// TwinCAT 3 PLC project Library
// Title: PMPS
// Company: SLAC - LCLS
// Author: Alex Wallace and contributors
// ProjectVersion: 0.0.0
// Description: Collection of PMPS functionality for LCLS PLCs
// ProgramVersion: 3.1.4023.0
// libraries:
//   Tc2_MC2, * (Beckhoff Automation GmbH)
//   Tc2_Standard, * (Beckhoff Automation GmbH)
//   Tc2_System, * (Beckhoff Automation GmbH)
//   Tc2_Utilities, * (Beckhoff Automation GmbH)
//   Tc3_JsonXml, * (Beckhoff Automation GmbH)
//   Tc3_Module, * (Beckhoff Automation GmbH)
//   LCLS General,newest,SLAC
//   TcUnit,newest,www.tcunit.org
// project tree:
//   DUTs/ E_BPTMState.TcDUT, K_Apertures.TcTLEO (not stored), L_Apertures.TcTLEO (not stored), L_Stopper.TcTLEO, K_Stopper.TcTLEO (not stored), ST_BeamParams_WC.TcDUT, ST_BeamParams.TcDUT, ST_Device.TcDUT (not stored), ST_DeviceState.TcDUT, ST_DeviceStateExt.TcDUT (not stored), ST_DeviceStateTable.TcDUT, ST_FFInfo.TcDUT, ST_FF.TcDUT, ST_FFOverride.TcDUT, ST_PMPS_Aperture.TcDUT, ST_PMPS_Attenuator.TcDUT, T_HashTableEntry.TcDUT (not stored)
//   GVLs/ PMPS_GVL.TcGVL
//   HelperFunctions/ APT_TO_IO.TcPOU (not stored), ATT_TO_IO.TcPOU (not stored), F_DeviceState_To_DeviceStateExt.TcPOU (not stored), F_DifferentBeamParams.TcPOU, F_eVRangeCalculator.TcPOU (not stored), F_eVWithinSpec.TcPOU, F_SafeBPCompare.TcPOU, F_SetBeamParams.TcPOU, F_SetStateParams.TcPOU (not stored), IO_TO_APT.TcPOU (not stored), IO_TO_ATT.TcPOU, IO_TO_BP.TcPOU, BP_TO_IO.TcPOU
//   / MAIN.TcPOU, PlcTask.TcTTO (not stored)
//   MajorComponents/Arbiter/ FB_Arbiter.TcPOU, FB_BeamParamAssertionPool.TcPOU
//   MajorComponents/ BeamParameterTransitionManager.TcPOU, FB_BPRequestor.TcPOU, FB_LinearDeviceStateTable.TcPOU, FB_LinearGovernor.TcPOU, I_HigherAuthority.TcIO
//   MajorComponents/FastFaults/ FB_FastFault.TcPOU, FB_FastFaultLogger.TcPOU, FB_HardwareFFOutput.TcPOU
//   MajorComponents/InterPlcComm/ FB_ArbiterToSubSys_IO.TcPOU, FB_SubSysToArbiter_IO.TcPOU
//   MajorComponents/PMPS_MPS_Interface/ FB_BeamClassOutputs.TcPOU, FB_CTLS_Outputs.TcPOU, FB_PhotonEnergyWatcher.TcPOU
//   TestComponents/ eBPTMTestStates.TcDUT (not stored), FB_Arbiter_Test.TcPOU, FB_AttenuatorSimulator.TcPOU (not stored), FB_BPTM_Test.TcPOU, FB_ArbToSubsys_Test.TcPOU, FB_DiffBP_Test.TcPOU (not stored), FB_SubsysToArb_Test.TcPOU, FB_evRangeCalculator_Test.TcPOU, FB_eVWithinSpec_Test.TcPOU (not stored), FB_FastFault_Test.TcPOU, FB_MachineSimulator.TcPOU, FB_PhotonEnergyWatcher_Test.TcPOU, FB_SafeBPCompare_Test.TcPOU, FB_SolidAttenuator.TcPOU (not stored) (excluded from build)
// real-time tasks:
//   TASK PlcTask: cycle T#10ms, priority 20, ADS port 350

// ---- DUTs/E_BPTMState.TcDUT
TYPE E_BPTMState :
(
	NewTarget := 1,
    WaitingForTransitionAssertion := 2,
    WaitingForFinalAssertion := 3,
    Transitioning := 4,
    CleaningUp := 5
);
END_TYPE

// ---- DUTs/L_Stopper.TcTLEO
{attribute 'qualified_only'}
{attribute 'strict'}
TYPE L_Stopper :
(
	ST1 := 1,
    ST2 := 2
);
END_TYPE

// ---- DUTs/ST_BeamParams_WC.TcDUT
TYPE ST_BeamParams_WC : 
    STRUCT
        (*  Requested pre-optic attenuation %  *)
		{attribute 'pytmc' := 'pv: Attenuation
        io: i'}
		fAtt : REAL := 100;
        (* Pulse-rate *)
        {attribute 'pytmc' := 'pv: Rate
        io: i'}
        nRate : UDINT := 10;
        (* Per pulse max energy (mJ) *)
        {attribute 'pytmc' := 'pv: PulseEnergy
        io: i'}
        fPP_mJ : REAL := 20;
        (* Photon energy ranges *)
        {attribute 'pytmc' := 'pv: PhotonEnergy
        io: i'}
        {attribute 'displaymode' := 'binary'}
        neVRange : WORD := 65535;
        (* Beamline attenuators *)
        {attribute 'pytmc' := 'pv: AuxAttenuator
        io: i'}
        astAttenuators : ARRAY [1..32] OF ST_PMPS_Attenuator;
        // Toggle for watchdog
        xValidToggle : BOOL;
        // Beam parameter set is valid (if readback), or acknowledged (if request)
        {attribute 'pytmc' := 'pv: Valid
        io: i'}
        xValid : BOOL;
        // Cohort index. Identifies which cohort this BP set was included in arbitration
        {attribute 'pytmc' := 'pv: Attenuation
        io: i'}
        nCohortInt : ULINT;
    END_STRUCT
END_TYPE

// ---- DUTs/ST_BeamParams.TcDUT
TYPE ST_BeamParams : 
    STRUCT
        (*  Requested pre-optic attenuation %  *)
		{attribute 'pytmc' := 'pv: Attenuation
            io: i
            field: EGU %
        '}
		fAtt : REAL := 100;
        (* Pulse-rate *)
        {attribute 'pytmc' := 'pv: Rate
            io: i
            field: EGU Hz
        '}
        nRate : UDINT := 10;
        (* Per pulse max energy (mJ) *)
        {attribute 'pytmc' := 'pv: PulseEnergy
            io: i
            field: EGU mJ
        '}
        fPP_mJ : REAL := 20;
        (* Photon energy ranges *)
        {attribute 'pytmc' := 'pv: PhotonEnergyRanges
            io: i
            field: EGU eV'}
        {attribute 'displaymode' := 'binary'}
        neVRange : WORD := 65535;
        (* Beamline attenuators *)
        {attribute 'pytmc' := 'pv: AuxAtt
        io: i'}
        astAttenuators : ARRAY [1..PMPS_GVL.AUX_ATTENUATORS] OF ST_PMPS_Attenuator;
        
        (* Stoppers *)
        {attribute 'pytmc' := 'pv: ST
        io: i'}
        aStoppers : ARRAY [1..PMPS_GVL.MAX_STOPPERS] OF BOOL;
        
        (* Apertures *)
        astApertures : ARRAY [1..PMPS_GVL.MAX_APERTURES] OF ST_PMPS_Aperture;
        
        // Toggle for watchdog
        xValidToggle : BOOL;
        // Beam parameter set is valid (if readback), or acknowledged (if request)
        {attribute 'pytmc' := 'pv: Valid
        io: i'}
        xValid : BOOL;
        // Cohort index. Identifies which cohort this BP set was included in arbitration
        {attribute 'pytmc' := 'pv: Cohort
        io: i
            field: DESC Cohort inc on each arb cycle
        '}
        nCohortInt : UDINT;
    END_STRUCT
END_TYPE

// ---- DUTs/ST_DeviceState.TcDUT
TYPE ST_DeviceState :
STRUCT
	
	//State name
	sStateName	:	STRING;
	nStateRef	:	UDINT; //Primary key of device state database
	
	//////////////////
	// This stuff may belong in a sub-class or something
	//Position
	rPosition	:	REAL := 0; //Center of the state
	//Tolerance
	rTolerance :	REAL := 0; //+/- amount
	//////////////////
	//Required beam parameters
	stReqBeamParam	:	ST_BeamParams;

END_STRUCT
END_TYPE

// ---- DUTs/ST_DeviceStateTable.TcDUT
TYPE ST_DeviceStateTable :
STRUCT
	iDeviceID:DINT;
	iStateID:DINT;
	rTargetPosition: REAL;
	rTolerance: REAL;
	rTransmission: REAL;
	iBeamClass : DINT;
	iPulseRate: DINT;
	rPerPulseEnergy:REAL;
	rUpper_eV: REAL;
	rLower_eV: REAL;
	rPhotonEnergy: REAL;
END_STRUCT
END_TYPE

// ---- DUTs/ST_FFInfo.TcDUT

// These elements should be set at init and never changed.

TYPE ST_FFInfo :
STRUCT
    sPath   :    T_MaxString; // Full PLC path to FF object
    Desc    :   T_MaxString; // Set at instantiation to a helpful description of the fast fault purpose
    DevName :   T_MaxString; // Component name, used in diagnostic to help narrow down where beam faults are coming from
    TypeCode    :   UINT; // Set at instantiation to fault class code

///////////////////////////////////////////
// Warning, this variable is effectively a VETO of the fast fault if set FALSE
// Do not alter the state of this variable unless you really know what you're doing.
///////////////////////////////////////////
    InUse   :   BOOL := FALSE; // If this FF is currently in-use
///////////////////////////////////////////

 
    AutoReset   :   BOOL; // Automatically clear fast fault (latching vs non-latching)
    
    {attribute 'pytmc' := '
        pv: InfoString
        io: i
     '}
    InfoString : STRING;
END_STRUCT
END_TYPE

// ---- DUTs/ST_FF.TcDUT
TYPE ST_FF :
STRUCT
    {attribute 'pytmc' := '
        pv: Info
     '}
    Info : ST_FFInfo;
    
    {attribute 'pytmc' := '
        pv: Veto
     '}
    Veto : ST_FFVeto;
    
    {attribute 'pytmc' := '
        pv: OK
        io: i
     '}
    OK   :   BOOL; // Fault logic state
    
    FaultAck : BOOL; // Set when faulted, reset by logger.
    
    {attribute 'pytmc' := '
        pv: BeamPermitted
        io: i
     '}
    BeamPermitted   :   BOOL; // Result of reset, veto, and fault logic, true beam off boolean
    
    {attribute 'pytmc' := '
        pv: Reset
        io: o
     '}
    Reset   :   BOOL;
    
    bsFF    :    RS;
    rtReset    :    R_TRIG;
    ftCountFault : F_TRIG;
    
END_STRUCT
END_TYPE

// ---- DUTs/ST_FFOverride.TcDUT
TYPE ST_FFOverride :
STRUCT
    {attribute 'pytmc' := '
        pv: Duration
        io: o
     '}
    Duration : UDINT; // UDINT to be compatible with ESS module.
    
    {attribute 'pytmc' := '
        pv: Activate
        io: o
     '}
    Activate : BOOL;
    
    {attribute 'pytmc' := '
        pv: Deactivate
        io: o
     '}
    Deactivate : BOOL;
    
    {attribute 'pytmc' := '
        pv: ElapsedTime
        io: i
     '}
    ElapsedTime : UDINT; // UDINT to be compatible with ESS module.
    
    {attribute 'pytmc' := '
        pv: Active
        io: i
     '} 
	Active: BOOL;
    
    Timer    :   TP;
    OvrdActLogAck : BOOL;
    OvrdExpLogAck : BOOL;
    
    tOvrdActivate : R_TRIG;
    tOvrdExpiring  : F_TRIG;
END_STRUCT
END_TYPE

// ---- DUTs/ST_PMPS_Aperture.TcDUT
TYPE ST_PMPS_Aperture :
STRUCT
    {attribute 'pytmc' := 'pv: Width
            io: i
            field: EGU mm'}
    Width : REAL; // distance between horizontal slits (x)
    {attribute 'pytmc' := 'pv: Height
            io: i
            field: EGU mm'}
    Height : REAL; // distance between vertical slits (y)
    
    {attribute 'pytmc' := 'pv: OK
        io: i'}
    xOK : BOOL; // status of aperture, false if error or in motion
END_STRUCT
END_TYPE

// ---- DUTs/ST_PMPS_Attenuator.TcDUT
TYPE ST_PMPS_Attenuator EXTENDS ST_PMPS_Attenuator_IO :
STRUCT
    (*
        {attribute 'pytmc' := 'pv: Att
            io: i
            field: EGU %
        '}
		nAtt : UINT;
        {attribute 'pytmc' := 'pv: OK
            io: i
        '}
		xAttOK : UINT; // true = no errors and attenuator is stable
        *)
END_STRUCT
END_TYPE

// ---- GVLs/PMPS_GVL.TcGVL
{attribute 'qualified_only'}
VAR_GLOBAL
    {attribute 'pytmc' := '
        pv: @(PREFIX)RequestedBP
        archive: 1Hz monitor
    '}
    stRequestedBeamParameters    :    ST_BeamParams; //Summarized request for the line, as recognized by the line arbiter PLC
    {attribute 'pytmc' := '
        pv: @(PREFIX)CurrentBP
        archive: 1Hz monitor
    '}
    stCurrentBeamParameters    :    ST_BeamParams; //Currently active BP set, broadcast by the line arbiter PLC
    
    fbLog : FB_LogMessage:=(eSubsystem:=E_Subsystem.MPS);
END_VAR
VAR_GLOBAL RETAIN    
    // Statistics
    {attribute 'pytmc' := '
        pv: @(PREFIX)SuccessfulPreemptions
        io: i
    '}
    SuccessfulPreemption : UDINT; // Any time BPTM applies a new BP request which is confirmed
    {attribute 'pytmc' := '
        pv: @(PREFIX)AccumulatedFastFaults
        io: i
    '}
    AccumulatedFF : UDINT; // Any time a FF occurs
END_VAR
VAR_GLOBAL CONSTANT
    EXCLUDED_ASSERTION_ID    :    UDINT    := 16#FFFFFFFF; //An assertion ID that should always return "not found" in the assertion pool
    VISIBLE_TEST_VELOCITY    :    LREAL    := 10;
    FAST_TEST_VELOCITY        :    LREAL    := 100;
    MAX_DEVICE_STATES        :    UDINT    := 300;
    MAX_FAST_FAULTS : UINT := 50; // Maximum number of fast faults that can be associated with a FFO
    MAX_STOPPERS    :   UINT := 16;
    {attribute 'pytmc' := '
        pv: @(PREFIX)FullBeamCnst
        archive: 1Hz monitor
        field: DESC Full beam constant
    '}    
    cstFullBeam    :    ST_BeamParams := (
        fAtt := 0,
        fPP_mJ := 1E4,
        neVRange := 2#1111_1111_1111_1111,
        nRate    := UDINT#1000000
    );
    {attribute 'pytmc' := '
        pv: @(PREFIX)SafeBeamCnst
        archive: 1Hz monitor
        field: DESC Safe beam constant
    '} 
    cstSafeBeam    :    ST_BeamParams := (
        fAtt := 100,
        fPP_mJ := 0,
        neVRange := 0,
        nRate    := 0
    );
    cnMaxStateArrayLen : INT := 20;
    
    AUX_ATTENUATORS : UINT := 16; // Maximum # of attenuators in the PMPS
    MAX_APERTURES : UINT := 4; // Maximum # of power slits in the PMPS
    DUMMY_AUX_ATT_ARRAY : ARRAY [1..PMPS_GVL.AUX_ATTENUATORS] OF ST_PMPS_Attenuator;
    
    MAX_ASSERTIONS    :    UDINT := 20; //Maximum number of assertions permitted in the arbiter
    
    g_cBoundaries    :    INT    := 15;
    {attribute 'pytmc' := '
        pv: @(PREFIX)eVRangeCnst
        archive: 1Hz monitor
        field: DESC eV Range constants
        field: EGU keV
    '}
    g_areVBoundaries    :    ARRAY [0..g_cBoundaries]    OF    REAL    := [ 
    0.2,
    0.3,
    0.4,
    0.5,
    0.6,
    0.7,
    0.8,
    0.9,
    1.0,
    1.1,
    1.2,
    1.3,
    1.4,
    1.5,
    1.6,
    1.7
];


END_VAR

// ---- MajorComponents/I_HigherAuthority.TcIO
INTERFACE I_HigherAuthority

METHOD CheckRequest : BOOL
VAR_INPUT
    nReqID    :    DWORD;
END_VAR
END_METHOD

METHOD RequestBP : BOOL
VAR_INPUT
    nReqID    :    DWORD; //StateID of state requesting beam parameter set
    stReqBP        :    ST_BeamParams; //Requested beam params
END_VAR
END_METHOD

END_INTERFACE

// ---- HelperFunctions/F_DifferentBeamParams.TcPOU
{attribute 'obsolete' := 'Use Req and Readback BP structs instead.'} 
(*DEPRECATED Compares BeamParam1 to BeamParam2, if any parameters of BeamParam1 are different than BeamParam2
the result will be true. *)
FUNCTION F_DifferentBeamParams : BOOL
VAR_INPUT
    BeamParam1    :    ST_BeamParams;
    BeamParam2    :    ST_BeamParams;
END_VAR
VAR
    // Internal Attenuation OK boolean
    xAttOK: BOOL := FALSE;
    // Internal Per-pulse energy OK boolean
    xPPmjOK: BOOL := FALSE;
    // Internal photon energy OK boolean
    xEvOK: BOOL := FALSE;
    xRateOK: BOOL;
END_VAR

xAttOK := BeamParam1.fAtt <> BeamParam2.fAtt;
xPPmjOK := BeamParam1.fPP_mJ <> BeamParam2.fPP_mJ;
xEvOK := BeamParam1.neVRange <> BeamParam2.neVRange;
xRateOK     := BeamParam1.nRate <> BeamParam2.nRate;


F_DifferentBeamParams := xAttOK OR xPPmjOK OR xEvOK OR xRateOK;

END_FUNCTION

// ---- HelperFunctions/F_eVWithinSpec.TcPOU
//reV must be within permitted range.
FUNCTION F_eVWithinSpec : BOOL
VAR_INPUT
    reV    :    REAL;    //Photon energy to check if within permitted range
    nPermittedRange    :    WORD; //Permitted range
END_VAR
VAR
    //Holding register for permitted ranges
    nPermittedRangeHolding    :    WORD; 
    //For loop counter
    nIndex    :    INT;
    // Lower boundary for range check 
    rPreviousBoundary: REAL := 0;
END_VAR

(* How this works:
The within range bool is initialized to false.
Load the word representation of ranges into a holding register.
If the bit at position zero of the holding register is true, and the input eV is
below the boundary at the index position of the boundary array, and the previous boundary
(which initializes at 0), then the within range bool is set. 
Then, we stash the upper boundary as the lower boundary for the next comparison,
and shift the holding register right, which moves the next bit to the zero position.
*)
nPermittedRangeHolding := nPermittedRange;

FOR nIndex := 0 TO PMPS_GVL.g_cBoundaries DO
        
    F_eVWithinSpec S= nPermittedRangeHolding.0 AND( 
        (reV <= PMPS_GVL.g_areVBoundaries[nIndex]*1000) AND
        (reV >= rPreviousBoundary*1000) );
        
    IF F_eVWithinSpec THEN RETURN; END_IF
    
    rPreviousBoundary := PMPS_GVL.g_areVBoundaries[nIndex];
    nPermittedRangeHolding := SHR(nPermittedRangeHolding, 1);
END_FOR

END_FUNCTION

// ---- HelperFunctions/F_SafeBPCompare.TcPOU
(*Compares BeamParam1 to BeamParam2: if the parameters of BeamParam1 are more conservative than BeamParam2
the result will be true. *)
FUNCTION F_SafeBPCompare : BOOL
VAR_INPUT
    BeamParam1    :    ST_BeamParams; //Must be more conservative than 2
    BeamParam2    :    ST_BeamParams;
END_VAR
VAR
    // Internal Attenuation OK boolean
    xAttOK: BOOL := FALSE;
    // Internal Per-pulse energy OK boolean
    xPPmjOK: BOOL := FALSE;
    // Internal photon energy OK boolean
    xEvOK: BOOL := FALSE;
    // Internal Beam Rate OK boolean
    xRateOK: BOOL;
    // Beam-rate is zero, masks all others considerations.
    xZeroRate: BOOL;
    
    idx : UINT;
    xAuxAttOK : BOOL;
    xAuxAprtOK : BOOL; 
END_VAR


xAttOK := BeamParam1.fAtt >= BeamParam2.fAtt;
xPPmjOK := BeamParam1.fPP_mJ <= BeamParam2.fPP_mJ;
xEvOK := (BeamParam1.neVRange AND BeamParam2.neVRange) = BeamParam1.neVRange;
xZeroRate    := BeamParam1.nRate = 0;
xRateOK    := BeamParam1.nRate <= BeamParam2.nRate;

FOR idx:=1 to PMPS_GVL.AUX_ATTENUATORS DO
    xAuxAttOK := BeamParam1.astAttenuators[idx].nAtt >= BeamParam2.astAttenuators[idx].nAtt;    
END_FOR

FOR idx:=1 to PMPS_GVL.MAX_APERTURES DO
    xAuxAprtOK := BeamParam1.astApertures[idx].Height <= BeamParam2.astApertures[idx].Height and
    BeamParam1.astApertures[idx].Width <= BeamParam2.astApertures[idx].Width;
END_FOR

F_SafeBPCompare := xZeroRate OR (xAttOK AND xPPmjOK AND xEvOK AND xRateOK AND xAuxAprtOK AND xAuxAttOK);

END_FUNCTION

// ---- HelperFunctions/F_SetBeamParams.TcPOU
FUNCTION F_SetBeamParams : ST_BeamParams
VAR_INPUT
    fAtt    :    REAL := 100;
    fPP_mJ: REAL := 0;
    neVRange    :    WORD := 0;
    nRate    :    UDINT := 0;
END_VAR
VAR
    BeamParams    :    ST_BeamParams;
    
END_VAR

BeamParams.fAtt := LIMIT(0,fAtt,100);
BeamParams.fPP_mJ := LIMIT(0,fPP_mJ,20);
BeamParams.neVRange := neVRange;
BeamParams.nRate    := MIN(nRate,1000000);

F_SetBeamParams    := BeamParams;

END_FUNCTION

// ---- HelperFunctions/IO_TO_ATT.TcPOU
FUNCTION IO_TO_ATT : ST_PMPS_Attenuator
VAR_INPUT
    IO : ST_PMPS_Attenuator_IO;
END_VAR
VAR
END_VAR

IO_TO_ATT.nAtt := IO.nAtt;
IO_TO_ATT.xAttOK := IO.xAttOK;

END_FUNCTION

// ---- HelperFunctions/IO_TO_BP.TcPOU
FUNCTION IO_TO_BP : ST_BeamParams
VAR_INPUT
    IO : ST_BeamParams_IO;
END_VAR
VAR
    idx : UINT;
END_VAR


FOR idx := 1 TO PMPS_GVL.AUX_ATTENUATORS DO
    IO_TO_BP.astAttenuators[idx] := IO_TO_ATT(IO.astAttenuators[idx]);
END_FOR

FOR idx := 1 TO PMPS_GVL.MAX_APERTURES DO
    IO_TO_BP.astApertures[idx] := IO_TO_APT(IO.astApertures[idx]);
END_FOR

IO_TO_BP.aStoppers := IO.aStoppers;
IO_TO_BP.fAtt := IO.fAtt;
IO_TO_BP.fPP_mJ := IO.fPP_mJ;
IO_TO_BP.nCohortInt := ULINT_TO_UDINT(IO.nCohortInt);
IO_TO_BP.neVRange := IO.neVRange;
IO_TO_BP.nRate := IO.nRate;
IO_TO_BP.xValid := IO.xValid;
IO_TO_BP.xValidToggle := IO.xValidToggle;

END_FUNCTION

// ---- HelperFunctions/BP_TO_IO.TcPOU
FUNCTION BP_TO_IO : ST_BeamParams_IO
VAR_INPUT
    BP : ST_BeamParams;
END_VAR
VAR
    idx : UINT := 0;
END_VAR


FOR idx := 1 TO PMPS_GVL.AUX_ATTENUATORS DO
    BP_TO_IO.astAttenuators[idx] := ATT_TO_IO(BP.astAttenuators[idx]);
END_FOR

BP_TO_IO.aStoppers := BP.aStoppers;
BP_TO_IO.fAtt := BP.fAtt;
BP_TO_IO.fPP_mJ := BP.fPP_mJ;
BP_TO_IO.nCohortInt := ULINT_TO_UDINT(BP.nCohortInt);
BP_TO_IO.neVRange := BP.neVRange;
BP_TO_IO.nRate := BP.nRate;
BP_TO_IO.xValid := BP.xValid;
BP_TO_IO.xValidToggle := BP.xValidToggle;

END_FUNCTION

// ---- MAIN.TcPOU
PROGRAM MAIN
VAR
    fbDiffBPTest    :    FB_DiffBP_Test;
    fbBPTMTest    :    FB_BPTM_Test;
    //fbSafeBPCompareTest    :    FB_SafeBPCompare_Test;
    //fbevWithinSpecTest    :    FB_evWithinSpec_Test;
    //fbPEWTest    :    FB_PhotonEnergyWatcher_Test;
    fbFFTest    :    FB_FastFault_Test;
    fbArbiterTest    :    FB_Arbiter_Test;
    //fbevRangeCalcTest : FB_evRangeCalculator_Test;
    fbSubSysToArbTest : FB_SubsysToArb_Test;
    fbArbToSubSysTest : FB_ArbToSubsys_Test;
END_VAR

TcUnit.RUN();

END_PROGRAM

// ---- TestComponents/FB_BPTM_Test.TcPOU
{attribute 'call_after_init'}
FUNCTION_BLOCK FB_BPTM_Test EXTENDS TcUnit.FB_TestSuite
VAR_INPUT
END_VAR
VAR_OUTPUT
END_VAR
VAR
END_VAR

BPTMBasicFunction();

METHOD BPTMBasicFunction
VAR_INPUT
END_VAR
VAR    
    //Final and transition assertions
    nTransitionID    :    UDINT := 1;
    stTransitionAssertion    :    ST_BeamParams := PMPS_GVL.cstSafeBeam;
    
     nReqID    :    UDINT    := 2;
    stReqAssertion    :    ST_BeamParams := PMPS_GVL.cstSafeBeam;
    
    fbMachine    :    FB_MachineSimulator;    
    
END_VAR
VAR_INST
    fbBPTM_TestBasicFunction    :    BeamParameterTransitionManager;
    fbArbiter    :    FB_Arbiter(1);
    xFirstPass    :    BOOL := TRUE;
    eTestStep: eBPTMTestStates := eBPTMTestStates.Init;
END_VAR
CASE eTestStep OF

eBPTMTestStates.Init:
    
    TEST('BPTMTest');
    eTestStep := eBPTMTestStates.WaitingForTransitionAssertion;

eBPTMTestStates.WaitingForTransitionAssertion:
    TEST('BPTMBasicFunction');
    
    //Call BPTM with requested final state and transition state
    fbBPTM_TestBasicFunction(
        fbArbiter := fbArbiter,
        i_TransitionAssertionID := nTransitionID,
        i_stTransitionAssertion := stTransitionAssertion,
        
        i_nRequestedAssertionID := nReqID,
        i_stRequestedAssertion := stReqAssertion
    );
    
    IF fbBPTM_TestBasicFunction.eBPTMState = E_BPTMState.WaitingForTransitionAssertion THEN
    
        AssertTrue(fbArbiter.CheckRequest(nTransitionID), 'Arbiter did not accept BPTM transition assertion');
        
        AssertFalse(fbArbiter.CheckRequest(nReqID), 'Arbiter has requested too early.');
                
        AssertFalse(fbBPTM_TestBasicFunction.q_xTransitionAuthorized,
            'Transition should not be authorized until the arbiter has final assertion');
            
        TEST_FINISHED_NAMED('BPTMBasicFunction');
        
        eTestStep := eBPTMTestStates.WaitingForFinalAssertion;
    END_IF

eBPTMTestStates.WaitingForFinalAssertion:

    TEST('BPTM Requests Final');
    fbBPTM_TestBasicFunction(fbArbiter := fbArbiter,
        stCurrentBeamParameters := stTransitionAssertion);
    
    IF fbBPTM_TestBasicFunction.eBPTMState = E_BPTMState.WaitingForFinalAssertion THEN
    
        AssertTrue(fbArbiter.CheckRequest(nReqID),
            'Transition assertion should be in arbiter');
        
        AssertTrue(fbArbiter.CheckRequest(nReqID),
            'Final assertion should be in arbiter');
            
        AssertFalse(fbBPTM_TestBasicFunction.q_xTransitionAuthorized,
            'Transition should not be authorized until the arbiter has final assertion');
            
        TEST_FINISHED_NAMED('BPTM Requests Final');
    
        eTestStep := eBPTMTestStates.Transitioning;
    END_IF

eBPTMTestStates.Transitioning:
    TEST('BPTM Authorizes Transition');
    fbBPTM_TestBasicFunction(fbArbiter := fbArbiter,
        stCurrentBeamParameters := stTransitionAssertion);
        
    IF fbBPTM_TestBasicFunction.eBPTMState = E_BPTMState.Transitioning THEN
    
        AssertTrue(fbArbiter.CheckRequest(nReqID),
            'Transition assertion should be in arbiter');
        
        AssertTrue(fbArbiter.CheckRequest(nReqID),
            'Final assertion should be in arbiter');
            
        AssertTrue(fbBPTM_TestBasicFunction.q_xTransitionAuthorized,
            'Transition should be authorized at this point.');
            
        AssertEquals(nReqID, fbBPTM_TestBasicFunction.nCurrentAssertionID,
            'nCurrentAssertionID not set.');
    
        TEST_FINISHED_NAMED('BPTM Authorizes Transition');
        
        eTestStep := eBPTMTestStates.CleaningUp;
    END_IF

eBPTMTestStates.CleaningUp:
    TEST_FINISHED_NAMED('BPTMTest');    
    
END_CASE
END_METHOD

END_FUNCTION_BLOCK

// ---- TestComponents/FB_MachineSimulator.TcPOU
(* Simulates the machine responding to requests by adding a bit of delay/ ramps
*)
FUNCTION_BLOCK FB_MachineSimulator
VAR_INPUT
    i_stAssertedParams    :    ST_BeamParams;
    i_xFault    :    BOOL;
END_VAR
VAR_OUTPUT
    q_stMachineParams    :    ST_BeamParams;
END_VAR
VAR
    fTargetAtt: REAL;
    tonAttTimer    :    TON := (
        PT := T#2S
        );
    fTargetPP_mJ: REAL;
    tonPPETimer: TON := (
        PT := T#2S
    );
END_VAR


//Attenuation
IF i_stAssertedParams.fAtt <> fTargetAtt THEN
    tonAttTimer(IN:=FALSE);
    fTargetAtt := i_stAssertedParams.fAtt;
ELSIF NOT tonAttTimer.Q THEN
    tonAttTimer(IN:=TRUE);
ELSE
    q_stMachineParams.fAtt := fTargetAtt;
END_IF

//Pulse Energy
IF i_stAssertedParams.fPP_mJ <> fTargetPP_mJ THEN
    tonPPETimer(IN:=FALSE);
    fTargetPP_mJ := i_stAssertedParams.fPP_mJ;
ELSIF NOT tonAttTimer.Q THEN
    tonPPETimer(IN:=TRUE);
ELSE
    q_stMachineParams.fPP_mJ := fTargetPP_mJ;
END_IF

//Rate
IF i_xFault THEN
    q_stMachineParams.nRate := 0;
ELSE
    q_stMachineParams.nRate := i_stAssertedParams.nRate;
END_IF

END_FUNCTION_BLOCK

// ---- MajorComponents/BeamParameterTransitionManager.TcPOU
(*
Implements the procedure for safely transitioning between device states by asserting the correct beam parameters for 
the state *)
FUNCTION_BLOCK BeamParameterTransitionManager
VAR_IN_OUT
    
    fbArbiter    :    FB_Arbiter; //Connect to local arbiter
    
END_VAR
VAR_INPUT
    i_TransitionAssertionID    :    UDINT := 0;
    i_stTransitionAssertion : ST_BeamParams := PMPS_GVL.cstSafeBeam; //Assertion required during transition (always safer than anything inbetween)
    
    i_nRequestedAssertionID    :    UDINT := 0;
    i_stRequestedAssertion    :    ST_BeamParams := PMPS_GVL.cstSafeBeam; //Requested assertion, change whenever
    
    i_xMoving    :    BOOL := FALSE; //Provide rising edge when device begins moving <remove>
    i_xDoneMoving    :    BOOL := FALSE; //Provide rising edge when device is done with a move
    
    stCurrentBeamParameters    :    ST_BeamParams := PMPS_GVL.cstFullBeam; //Connect to current beam parameters
    
END_VAR
VAR_OUTPUT

    q_xTransitionAuthorized    :    BOOL := FALSE; //Rising edge indicating the device is safe to move, use as input to move execute (which requires a rising edge)

END_VAR

VAR
    nTargetAssertionID    :    UDINT := 0;
    stTargetAssertion    :    ST_BeamParams; //Current target assertion
    nCurrentAssertionID    :    UDINT := 0;
    
    xNewBP    :    BOOL;
    xTranBP    :    BOOL;
    xFinalBP    :    BOOL;
    
    eBPTMState : E_BPTMState;
    ePrevState : E_BPTMState;
    
    xEntry : BOOL;
    rTransition : R_TRIG;
    xNewTarget : BOOL;
    
END_VAR


// Execute exit actions before transition back to NewTarget
IF nTargetAssertionID <> i_nRequestedAssertionID THEN
    CASE eBPTMState OF
        //NewTarget:
        WaitingForTransitionAssertion:
            WaitingForTransitionAssertion_EXIT();
        WaitingForFinalAssertion:
            WaitingForFinalAssertion_EXIT();
        Transitioning:
            DeauthorizeTransition();
        //CleaningUp: 
	END_CASE
    
    eBPTMState := E_BPTMState.NewTarget;
    
END_IF

xEntry S= ePrevState <> eBPTMState;

// States
CASE eBPTMState OF
    NewTarget:
        IF xEntry THEN
            NewTarget_ENTRY();
        ELSIF xNewBP THEN
            eBPTMState := E_BPTMState.WaitingForTransitionAssertion;
        ELSE
            SetNewTarget();
        END_IF
            
    WaitingForTransitionAssertion:
        IF xEntry THEN
            AssertTransitionBP();
        ELSIF xTranBP THEN
            WaitingForTransitionAssertion_EXIT();
            eBPTMState := E_BPTMState.WaitingForFinalAssertion;
        ELSE
            WaitingForTransitionAssertion_DO();
        END_IF
        
    WaitingForFinalAssertion:
        IF xEntry THEN
            AssertFinalBP();
        ELSIF xFinalBP THEN
            WaitingForFinalAssertion_EXIT();
            eBPTMState := E_BPTMState.Transitioning;
        ELSE
            WaitingForFinalAssertion_DO();
        END_IF
        
    Transitioning:
        IF xEntry THEN
            AuthorizeTransition();
        ELSIF i_xDoneMoving THEN
            DeauthorizeTransition();
            eBPTMState := E_BPTMState.CleaningUp;
		END_IF
        
    CleaningUp:
        IF xEntry THEN
            RemoveTransitionAssertion();
		END_IF
END_CASE

ePrevState := eBPTMState;

ACTION AssertFinalBP:
//q_stFinalAssertion := stTargetAssertion;

//Clearing previous target parameters
(* This is considered safe at this step as the transition
state beam parameters should always be safer than the
current or target state beam parameters
*)
fbArbiter.RemoveRequest( nCurrentAssertionID );

//Asserting target parameters
fbArbiter.AddRequest(
    nTargetAssertionID,
    stTargetAssertion
);

//Remembering final assertionID for removal later
nCurrentAssertionID := nTargetAssertionID;
END_ACTION

ACTION AssertTransitionBP:

fbArbiter.AddRequest(
    i_TransitionAssertionID,
    i_stTransitionAssertion
);
END_ACTION

ACTION AuthorizeTransition:
q_xTransitionAuthorized := TRUE;
END_ACTION

ACTION DeauthorizeTransition:
q_xTransitionAuthorized := FALSE;
END_ACTION

ACTION NewTarget_ENTRY:
xNewBP := False;
END_ACTION

ACTION RemoveTransitionAssertion:
//q_stTransitionAssertion := PMPS_GVL.cstFullBeam;

//Removing transition assertion
fbArbiter.RemoveRequest( i_TransitionAssertionID );



//TODO add something to verify removal
END_ACTION

ACTION SetNewTarget:
IF i_nRequestedAssertionID <> 0 AND
    i_nRequestedAssertionID <> PMPS_GVL.EXCLUDED_ASSERTION_ID THEN
    
    stTargetAssertion := i_stRequestedAssertion;
    nTargetAssertionID := i_nRequestedAssertionID;
    xNewBP := TRUE;
END_IF
END_ACTION

ACTION WaitingForFinalAssertion_DO:
//Final Assertion Verification

xFinalBP := F_SafeBPCompare(stCurrentBeamParameters, stTargetAssertion) AND
    fbArbiter.CheckRequest( i_nRequestedAssertionID);;
END_ACTION

ACTION WaitingForFinalAssertion_EXIT:
//Set this bool false so we can get a rising edge on the next try
xFinalBP := FALSE;
PMPS_GVL.SuccessfulPreemption := PMPS_GVL.SuccessfulPreemption + 1;
END_ACTION

ACTION WaitingForTransitionAssertion_DO:
//Transition Assertion Verification
xTranBP    := F_SafeBPCompare(stCurrentBeamParameters, i_stTransitionAssertion) AND
    fbArbiter.CheckRequest(i_TransitionAssertionID);
END_ACTION

ACTION WaitingForTransitionAssertion_EXIT:
xTranBP := FALSE;
PMPS_GVL.SuccessfulPreemption := PMPS_GVL.SuccessfulPreemption + 1;
END_ACTION

END_FUNCTION_BLOCK

// ---- MajorComponents/Arbiter/FB_Arbiter.TcPOU
(* FB Arbiter

The arbiter primary objectives are:
- Provide a simple interface for devices to request beam parameter sets
- Provide a way for devices to verify their BPS is active in the arbiter
- Provide a way for devices remove their requests from evaluation
- Evaluate all active beam parameter requests registered with the aribiter,
to determine the safest combination of all sets, provide this set as an output.
- Do all of this with minimal overhead

To these ends, the arbiter uses a hash-table, the rows being a state-id as the key, and a corresponding
 beam parameter set to be evaluated against all the other sets (or rows), in the table.
 
The hash table can be thought of as an array on steriods, they are worth reading about, suffice to say
the hash table will tell you when you reach the end of all the entries, and enables us to find entries quickly.

These features efficiently address the addition, removal, and verification of beam parameter sets listed in the above requirements.

An important thing to pay attention to is the A_Arbitrate action. This action implements the evaluation of beam parameter
sets against each other.

*)

FUNCTION_BLOCK FB_Arbiter
VAR_INPUT
END_VAR
VAR_OUTPUT
    {attribute 'pytmc' := '
        pv: ArbitratedBP
        io: i
        field: DESC Arbitrated BP
     '}
    q_stBeamParams    :    ST_BeamParams; //Updated on each cycle of the arbiter FB with the current arbitrated beam parameter set
    
    q_xStateIDFound    :    BOOL; //Set true if a state-id is found in the assertion pool after calling A_VerifyAssertion
END_VAR
VAR
    {attribute 'pytmc' := '
        pv: AP
        io: i
        field: DESC Assertion Pool
     '}
    fbBPAssertionPool    :    FB_BeamParamAssertionPool; //Table of active beam parameter assertions

    xRequestMade : BOOL; // Arbiter has confirmed its request has made it into the beam parameter request    
    
    {attribute 'pytmc' := '
        pv: ArbiterID
        io: i
        field: DESC Arbiter ID for elev. req.
     '}
    nArbiterID : UDINT; // Arbiter ID, used for making higher-level BP requests
    {attribute 'pytmc' := '
        pv: CohortCounter
        io: i
        field: DESC Intrnl cohort counter
     '}
    nArbiterCohort : UDINT := 1; // The cohort index keeps track of which beam parameter requests have been included in higher-level arbitrations
    // Init to 1, provides a guard against default cohort value in BP requests.
    {attribute 'pytmc' := '
        pv: ActiveInArbitration
        io: i
        field: DESC True if this arbiter's req is included
     '}
    xActiveInArbitration : BOOL; // True when this arbiter's request is included in all higher-level arbitrations
END_VAR

METHOD AddRequest : BOOL
VAR_INPUT
    nReqID    :    DWORD; //StateID of state requesting beam parameter set
    stReqBP        :    ST_BeamParams; //Requested beam params
END_VAR
VAR_INST
    fbLog : FB_LogMessage;
END_VAR
// If the request is already in the pool, then skip the rest.
// This is flawed, needs to update the request if it's already in the pool, despite having the same ID
IF THIS^.CheckRequestInPool(nReqID) THEN
    AddRequest := FALSE;
    RETURN;
END_IF

IF nReqID <> PMPS_GVL.EXCLUDED_ASSERTION_ID THEN
    stReqBP.nCohortInt := nArbiterCohort; // Set the cohort number for this BP request.
    
    THIS^.fbBPAssertionPool.A_Add(
        key := nReqID,
        putValue := stReqBP
    );
END_IF
    
IF NOT THIS^.fbBPAssertionPool.bOk THEN
    fbLog(sMsg:='Addition to arbiter assertion pool failed',
            eSevr:=TcEventSeverity.Warning,
            eSubsystem:=E_Subsystem.MPS);
END_IF

// With any new request reset the internal arbiter "done" flag
xRequestMade := FALSE;

AddRequest := THIS^.fbBPAssertionPool.bOk;
END_METHOD

METHOD ArbitrateBP : ST_BeamParams
VAR_INPUT
    stBP1    :    ST_BeamParams;
    stBP2    :    ST_BeamParams;
END_VAR
VAR
    idx : UINT := 1;
END_VAR
//<TODO>Add something here to register the key that won for each param

//Attenuation
ArbitrateBP.fAtt := MAX(stBP1.fAtt, stBP2.fAtt);

FOR idx := 1 TO PMPS_GVL.AUX_ATTENUATORS DO
    ArbitrateBP.astAttenuators[idx].nAtt := MAX(stBP1.astAttenuators[idx].nAtt, stBP2.astAttenuators[idx].nAtt);
END_FOR

//Apertures
FOR idx := 1 TO PMPS_GVL.MAX_APERTURES DO
    ArbitrateBP.astApertures[idx].Height := MIN(stBP1.astApertures[idx].Height, stBP2.astApertures[idx].Height);
    ArbitrateBP.astApertures[idx].Width := MIN(stBP1.astApertures[idx].Width, stBP2.astApertures[idx].Width);
END_FOR

//Pulse energy
ArbitrateBP.fPP_mJ := MIN(stBP1.fPP_mJ, stBP2.fPP_mJ);

//Photon energy ranges
ArbitrateBP.neVRange := stBP1.neVRange AND stBP2.neVRange;

//Rate
ArbitrateBP.nRate := MIN(stBP1.nRate, stBP2.nRate);
END_METHOD

(* Searches state assertion pool for a state-id, and sets q_xStateIDFound true if found.

Use like so:
IF fbArbiter.CheckRequest(nStateIDAssertionToCheck) THEN:
    Request is found and active in arbitration,. Do something.
ELSE:
    Request was not found, or is not yet included in arbitration. Don't do something/ wait.

*)
METHOD CheckRequest : BOOL
VAR_INPUT
    nReqID    :    DWORD;
END_VAR
VAR
    BP : ST_BeamParams;
END_VAR
fbBPAssertionPool.A_Lookup(key := nReqID);

// Verify BP is acknowledged
BP := fbBPAssertionPool.getValue;

// This logic:
// Did we find the assertion in the pool?
// Is the assertion cohort number less than the current cohort and greater than zero?
// Is the Aribter itself active in arbitration?
CheckRequest := fbBPAssertionPool.bOk AND 
                BP.nCohortInt < nArbiterCohort AND
                BP.nCohortInt > 0 AND 
                xActiveInArbitration;
END_METHOD

// Verify request is at least in the pool
// Does not verify request has been included in arbitration.
// Use CheckRequest instead.
METHOD CheckRequestInPool : BOOL
VAR_INPUT
    nReqID    :    DWORD;
END_VAR
THIS^.fbBPAssertionPool.A_Lookup(key := nReqID);

CheckRequestInPool := THIS^.fbBPAssertionPool.bOk;
END_METHOD

// Elevates the arbitrated BP set to something above.
// Could be another arbiter, or a BP requester/ IO, 
// or an FB that locks in a specific portion of the BP set.
METHOD ElevateRequest : BOOL
VAR_INPUT
    HigherAuthority : I_HigherAuthority;
END_VAR
(*
This method should only be used with one higher level component.
*)

IF NOT xRequestMade THEN
    xRequestMade := HigherAuthority.RequestBP(nReqID := nArbiterID, stReqBP := GetArbitratedBP());
    xActiveInArbitration := FALSE;
END_IF

IF HigherAuthority.CheckRequest(nReqID := nArbiterID) AND NOT xActiveInArbitration THEN // Check request must verify the ID is present and accounted for in arbitration
    nArbiterCohort := nArbiterCohort + 1; // This cohort number is for all subordinate requests within the arbiter
    xActiveInArbitration := TRUE;
END_IF
END_METHOD

METHOD FB_init : BOOL
VAR_INPUT
	bInitRetains : BOOL; // if TRUE, the retain variables are initialized (warm start / cold start)
	bInCopyCode : BOOL;  // if TRUE, the instance afterwards gets moved into the copy code (online change)
    nID : DWORD := PMPS_GVL.EXCLUDED_ASSERTION_ID; // Arbiter ID, must be globally unique.
END_VAR
nArbiterID := nId;
fbBPAssertionPool.A_Reset();
END_METHOD

METHOD GetArbitratedBP : ST_BeamParams
VAR_INPUT
END_VAR
VAR
    getPosPtr    : POINTER TO T_HashTableEntry := 0;
    getBPStruct    :    ST_BeamParams;
    
    stOutputBP    :    ST_BeamParams; //Holding struct for arbitration process
END_VAR
VAR_INST
    xFirstPass : BOOL := TRUE;
    fbGetCurTaskIdx : GETCURTASKINDEX;
    LastCycleCount : UDINT;
    fbLogMessage : FB_LogMessage;
END_VAR
//Arbitrate
(*
This step cycles through every hash table entry, comparing
the beam parameters from each assertion to what we're planning
to assert.

The safer of the two parameters is kept so at the end we may
have a mix of beam parameters, the composition being safe for
all asserters.

*)

THIS^.fbBPAssertionPool.A_GetFirst( putPosPtr := 0, getPosPtr=>getPosPtr, getValue=>getBPStruct );
IF THIS^.fbBPAssertionPool.bOk THEN //If the table is empty (not OK), we are left with the default stOutputBP set above.
    
    //The first entry in the hash table is taken as the setting to arbitrate against
    stOutputBP := F_SetBeamParams(
        fAtt := getBPStruct.fAtt,
        astAuxAtt := getBPStruct.astAttenuators,
        fPP_mJ := getBPStruct.fPP_mJ,
        neVRange    := getBPStruct.neVRange,
        nRate := getBPStruct.nRate
    );

    REPEAT
        THIS^.fbBPAssertionPool.A_GetNext( putPosPtr := THIS^.fbBPAssertionPool.getPosPtr, getPosPtr=>getPosPtr, getValue=>getBPStruct );
        IF THIS^.fbBPAssertionPool.bOk THEN
            stOutputBP := ArbitrateBP(stOutputBP, getBPStruct);
        END_IF
    UNTIL NOT fbBPAssertionPool.bOk
    END_REPEAT
ELSE
    //Safest parameters to start
    stOutputBP := PMPS_GVL.cstSafeBeam;
END_IF
(*
stOutputBP.AckInt := stOutputBP.AckInt + 1; // Arbitration cycle

// Verify this function hasn't been run twice this cycle
IF xFirstPass THEN
    fbGetCurTaskIdx();
END_IF

IF LastCycleCount <> _TaskInfo[fbGetCurTaskIdx.index].CycleCount THEN
    // Good
    LastCycleCount := _TaskInfo[fbGetCurTaskIdx.index].CycleCount;
ELSE
    fbLogMessage(i_sMsg := 'GetArbitratedBP run more than once in a cycle.',
        i_eSevr := E_MesgSevr.Error,
        i_eSubsystem := E_Subsystem.MPS);
END_IF
*)


q_stBeamParams := stOutputBP;

GetArbitratedBP.fAtt := stOutputBP.fAtt;
GetArbitratedBP.fPP_mJ := stOutputBP.fPP_mJ;
GetArbitratedBP.neVRange := stOutputBP.neVRange;
GetArbitratedBP.nRate := stOutputBP.nRate;

GetArbitratedBP.xValidToggle := NOT GetArbitratedBP.xValidToggle;

xFirstPass := FALSE;
END_METHOD

(* Searches for a state-id, and removes it from the assertion pool.

Use like so:
fbArbiter.A_RemoveAssertion(
i_nStateId := nStateIDAssertionToRemove
);

*)
METHOD RemoveRequest : BOOL
VAR_INPUT
    nReqId    :    DWORD;
END_VAR
IF nReqId <> PMPS_GVL.EXCLUDED_ASSERTION_ID THEN
    THIS^.fbBPAssertionPool.A_Remove(key := nReqId);
    
    IF THIS^.fbBPAssertionPool.bOk THEN
        ;
    ELSE
        ;
    END_IF
END_IF

RemoveRequest := THIS^.fbBPAssertionPool.bOk;
END_METHOD

END_FUNCTION_BLOCK

// ---- MajorComponents/Arbiter/FB_BeamParamAssertionPool.TcPOU
(* This function block implements simple database. Data element values are stored in the hash table.  *)
FUNCTION_BLOCK FB_BeamParamAssertionPool
VAR_INPUT
    key         : DWORD := 0;(* Entry key: used by A_Lookup, A_Remove method, the key variable is also used by A_Add method *)
    putPosPtr    : POINTER TO T_HashTableEntry := 0;(* Hash table entry position pointer (used by A_Find, A_GetNext, A_GetPrev) *)
    putValue     : ST_BeamParams;(* Hash table entry value (used by A_AddHead, A_AddTail, A_Find )*)
END_VAR
VAR_OUTPUT
    bOk            : BOOL := FALSE;(* TRUE = Success, FALSE = Failed *)
    getPosPtr    : POINTER TO T_HashTableEntry := 0;(* Returned hash table entry position pointer *)
    getValue     : ST_BeamParams;(* Returned hash table entry value *)
    nCount        : UDINT := 0;(* Hash table size (number of used entries, used by A_Count) *)
END_VAR
VAR
    {attribute 'pytmc' := '
        pv: Entry
        io: i
     '}
    dataPool    : ARRAY[0..PMPS_GVL.MAX_ASSERTIONS] OF ST_BeamParams;(* Structured data element pool *)
    {attribute 'pytmc' := '
        pv: Key
        io: i
     '}
    entries        : ARRAY[0..PMPS_GVL.MAX_ASSERTIONS] OF T_HashTableEntry;(* Max. number of hash table entries. The value of table entry = 32 bit integer (pointer to dataPool-array-entry) *)
    fbTable     : FB_HashTableCtrl;(* basic hash table control function block *)
    hTable         : T_HHASHTABLE;(* hash table handle *)
    pRefPtr        : POINTER TO ST_BeamParams := 0;
    indexOfElem    : ULINT;(* Integer value (max. size: x86=>32bit, x64=>64bit)*)
END_VAR

;

ACTION A_Add:
(* Adds entry to the table *)
MEMSET( ADR( getValue ), 0, SIZEOF( getValue ) );
getPosPtr := 0;

fbTable.A_Add( hTable := hTable, key := key, putValue := ADR(PMPS_GVL.cstSafeBeam)(* we will set this value later *), getPosPtr=>getPosPtr, bOk=>bOk );(* Add new element to the table, getPosPtr points to the new entry *)
IF fbTable.bOk THEN(* Success *)
    fbTable.A_GetIndexAtPosPtr( hTable := hTable, putPosPtr := getPosPtr, getValue =>indexOfElem, bOk=>bOk );(* Get array index of getPosPtr entry *)
    IF fbTable.bOk THEN(* Success *)
        pRefPtr     := ADR( dataPool[indexOfElem] );(* Get pointer to the data element *)

        pRefPtr^ := putValue;(* copy application value *)

        fbTable.A_Add( hTable := hTable, key := key, putValue := pRefPtr, bOk=>bOk );(* Assign the entry value = pointer to the data element *)
        IF fbTable.bOk THEN(* Success *)
            getValue := putValue;
        END_IF
    END_IF
END_IF
END_ACTION

ACTION A_Count:
(* Count number of used entries *)
nCount := hTable.nCount;
bOk := TRUE;
END_ACTION

ACTION A_GetFirst:
(* Get first entry position pointer and value *)
MEMSET( ADR( getValue ), 0, SIZEOF( getValue ) );
getPosPtr := 0;

fbTable.A_GetFirst( hTable := hTable, putPosPtr := putPosPtr, getValue=>pRefPtr, getPosPtr=>getPosPtr, bOk=>bOk );
IF fbTable.bOk THEN
    getValue := pRefPtr^;
END_IF
END_ACTION

ACTION A_GetNext:
(* Get next entry position pointer and value *)
MEMSET( ADR( getValue ), 0, SIZEOF( getValue ) );
getPosPtr := 0;
bOk := FALSE;

IF putPosPtr = 0 THEN
    RETURN;
END_IF

fbTable.A_GetNext( hTable := hTable, putPosPtr := putPosPtr, getValue=>pRefPtr, getPosPtr=>getPosPtr, bOk=>bOk );
IF fbTable.bOk THEN
    getValue := pRefPtr^;
END_IF
END_ACTION

ACTION A_Lookup:
(* Lookup for entry by key  *)
MEMSET( ADR( getValue ), 0, SIZEOF( getValue ) );
getPosPtr := 0;

fbTable.A_Lookup( key := key, hTable := hTable, putPosPtr := putPosPtr, getValue=>pRefPtr, getPosPtr=>getPosPtr, bOk=>bOk );
IF fbTable.bOk THEN
    getValue := pRefPtr^;
END_IF
END_ACTION

ACTION A_Remove:
(* Search for entry and remove it *)
MEMSET( ADR( getValue ), 0, SIZEOF( getValue ) );
getPosPtr := 0;

fbTable.A_Remove( key := key, hTable := hTable, putPosPtr := putPosPtr, getValue=>pRefPtr, getPosPtr=>getPosPtr, bOk=>bOk );
IF fbTable.bOk THEN
    getValue := pRefPtr^;
END_IF
END_ACTION

ACTION A_Reset:
(* Reset/initialize linked list *)
MEMSET( ADR( getValue ), 0, SIZEOF( getValue ) );
getPosPtr := 0;
bOk := F_CreateHashTableHnd( ADR( entries ), SIZEOF( entries ), hTable );(* Intialize table handle *)
fbTable.A_Reset( hTable := hTable, bOk=>bOk );
nCount := 0;
END_ACTION

END_FUNCTION_BLOCK

// ---- TestComponents/FB_FastFault_Test.TcPOU
{attribute 'call_after_init'}
FUNCTION_BLOCK FB_FastFault_Test EXTENDS TcUnit.FB_TestSuite
VAR_INPUT
END_VAR
VAR_OUTPUT
END_VAR
VAR

END_VAR

FFCombinedFunctionality();
FFRegistration();

METHOD FFCombinedFunctionality
VAR_INPUT
END_VAR
VAR_INST
    fbFF    :    FB_FastFault;
    fbFFO    :    FB_HardwareFFOutput;
    
END_VAR
TEST('FFCombinedFunctionality');

//Clear initial faults
fbFFO.i_xReset:=TRUE; //Reset requested at start of cycle

fbFF(io_fbFFHWO := fbFFO, //FF reset somehwere in code
    i_xOK := TRUE,
    i_xReset := TRUE);

fbFFO.EvaluateOutput(); //FFO eval called at end of cycle
    
AssertTrue(fbFFO.q_xFastFaultOut,
    'Fast fault did not clear');


//Induce fault with FF

fbFFO(i_xReset := FALSE); //Reset released at start of cycle

fbFF(io_fbFFHWO := fbFFO, //FF faulted
    i_xOK := FALSE); //Reset is still set true from last call.
    
fbFFO.EvaluateOutput(); //FFO eval called at end of cycle

AssertFalse(fbFFO.q_xFastFaultOut,
    'Fast fault did not trip the beam');
    
    
//FFO remains faulted until local (FF) and FFO receieve fresh reset request, and faults
//are actually cleared

//Attempt to clear FFO fails because FF still faulted
fbFFO.i_xReset := TRUE; //Reset requested

fbFF(io_fbFFHWO := fbFFO, //FF faulted
    i_xOK := FALSE,
    i_xReset := FALSE);
    
fbFFO.EvaluateOutput(); //FFO eval called at end of cycle

AssertFalse(fbFFO.q_xFastFaultOut,
    'Fast fault output cleared while fault remains, very bad');
    
//Attempt to clear FF while fault remains fails
fbFFO.EvaluateOutput(i_xReset := FALSE);

fbFFO.i_xReset := TRUE; //Reset requested

fbFF(io_fbFFHWO := fbFFO, //FF faulted
    i_xOK := FALSE,
    i_xReset := TRUE); //This reset should fail.
    
fbFFO.EvaluateOutput(); //FFO eval called at end of cycle

AssertFalse(fbFFO.q_xFastFaultOut,
    'Fast fault cleared while fault remains, very bad');
    
TEST_FINISHED();
END_METHOD

METHOD FFRegistration
VAR_INPUT
END_VAR
VAR_INST
    fbFF    :    FB_FastFault;
    fbFFO    :    FB_HardwareFFOutput;
END_VAR
TEST('FFRegistration');

fbFF(io_fbFFHWO := fbFFO);

AssertEquals_STRING(fbFF.sPath, fbFFO.astFF[fbFF.RegistrationIdx].Info.sPath,
    'FF registration with FFO did not succeed');

TEST_FINISHED();
END_METHOD

END_FUNCTION_BLOCK

// ---- MajorComponents/FastFaults/FB_FastFault.TcPOU
(* Fast Fault
2019-9-13 A. Wallace

Use this block to generate a beam-off fault. Connects to a fast fault hardware output 
function block to contribute to the state of the fast fault output (FFO).

If the i_xOK goes false, the associated FFO will go false, despite the state of any other
contributing fast faults, unless the FFO is currently vetoed.

*)
{attribute 'reflection'}
FUNCTION_BLOCK FB_FastFault
VAR_INPUT
    {attribute 'pytmc' := '
        pv: FastFaultInput
        io: i
     '}
    i_xOK        :    BOOL; // Connect to fast-fault condition (false produces fault)
    {attribute 'pytmc' := '
        pv: ResetFault
        io: o
     '}
    i_xReset    :    BOOL; // Resets when i_xOK is true and this is true
    {attribute 'pytmc' := '
        pv: AutoReset
        io: i
     '}
    i_xAutoReset : BOOL := FALSE; // Automatically clear fast fault (latching vs non-latching)
    
    i_DevName : T_MaxString := ''; // Device name for diagnostic
    i_Desc : T_MaxString := ''; // Description of fast fault (you should set at init)
    i_TypeCode : UINT; // Error code for classifying fast faults
END_VAR
VAR_OUTPUT
    {attribute 'pytmc' := '
        pv: FastFaultOK
        io: i
     '}
    o_xFFLine    :    BOOL; //Connect to HW output or another FF input if you like (Optional)
END_VAR
VAR_IN_OUT
    io_fbFFHWO        :    FB_HardwareFFOutput; //Point to FB_HardwareFFOutput of your choice
END_VAR
VAR
    {attribute 'instance-path'}
    {attribute 'noinit'}
    sPath    :    T_MaxString;
    
    FFInfo : ST_FFInfo;
    
    RegistrationIdx : UINT := 1; // The index this FF was registered in the FFO
    
    xInit    :    BOOL :=TRUE;
    
    InfoStringFmtr : FB_FormatString;
    
    InUse : T_MaxString;
    AutoReset : T_MaxString;

END_VAR

IF xInit    THEN
    FFInfo.sPath := sPath;
    FFInfo.InUse := True;
    FFInfo.TypeCode := i_TypeCode;
    FFInfo.DevName := i_DevName;
    FFInfo.Desc := i_Desc;
    FFInfo.AutoReset := i_xAutoReset;
    
    InUse := BOOL_TO_STRING(FFInfo.InUse);
    AutoReset := BOOL_TO_STRING(FFInfo.AutoReset);
    InfoStringFmtr(sFormat:='%s;%s;%X;%s;%s;%s;',
        arg1 := F_STRING(FFinfo.sPath),
        arg2 := F_STRING(InUse),
        arg3 := F_WORD(FFInfo.TypeCode),
        arg4 := F_STRING(FFInfo.DevName),
        arg5 := F_STRING(FFInfo.Desc),
        arg6 := F_STRING(AutoReset),
        sOut=>FFInfo.InfoString);
    io_fbFFHWO.Register(
        stFFInfo:=FFInfo, 
        Idx=>RegistrationIdx);
    //<TODO> if registration doesn't succeed, send warning to diagnostic
    xInit := FALSE;
END_IF

io_fbFFHWO.IdxCheckIn(Idx:=RegistrationIdx, OK := i_xOK, Reset:= i_xReset);

END_FUNCTION_BLOCK

// ---- MajorComponents/FastFaults/FB_HardwareFFOutput.TcPOU
{attribute 'reflection'}
FUNCTION_BLOCK FB_HardwareFFOutput
VAR CONSTANT
    FF_ARRAY_UPPER_BOUND : DINT := PMPS_GVL.MAX_FAST_FAULTS;
END_VAR
VAR_INPUT
    {attribute 'pytmc' := '
        pv: ClearFault
        io: o
     '}
    i_xReset    :    BOOL;
    {attribute 'pytmc' := '
        pv: EnableVeto
        io: o
     '}
    i_xVeto    :    BOOL;    
END_VAR
VAR_OUTPUT
    {attribute 'pytmc' := '
        pv: FaultHWO
        io: i
     '}
    q_xFastFaultOut    AT %Q*    :    BOOL;
END_VAR
VAR_IN_OUT

END_VAR
VAR
    {attribute 'pytmc' := '
        pv: FF
     '}
    astFF : ARRAY[1..FF_ARRAY_UPPER_BOUND] OF ST_FF;
    
    {attribute 'pytmc' := '
        pv: RegistrationFailure
        io: io
     '}
    xFastFaultRegFail  :   BOOL := FALSE; // Set true if a fast fault fails to register. Holds beam off.
    tFFRegFail : F_TRIG;
    
    {attribute 'instance-path'}
    {attribute 'noinit'}
    sPath    :    T_MaxString;

	{attribute 'pytmc' := '
        pv: OK
        io: i
     '}
    xOK    :    BOOL:= TRUE; // Current internal state of FFO, indicates if FFO will accept a reset
    
    rtReset    :    R_TRIG;
    rtResetandOK : R_TRIG;
    
    nIndex    :    UINT := 1;
	
	IdxOK: BOOL;
    
    
    fbJson : FB_JsonSaxWriter;
    pmpsTypeCode : UDINT := 0; // shows up in json as pmps_typecode
    fbLogger : FB_LogMessage := (
        eSevr := TcEventSeverity.Critical,
        eSubsystem := E_Subsystem.MPS);

END_VAR

// <TODO> latch off beam if DI card status goes bad

ACTION EvaluateOutput:

////////////////////////////////////////////////////////////////
// Critical code. Do not touch unless you know what you're doing
////////////////////////////////////////////////////////////////

//<TODO> add diagnostic for success or failure of reset
rtReset(CLK:=i_xReset);
rtResetandOK(CLK:=rtReset.Q AND xOK); // Need two R_TRIG to avoid autoreset

q_xFastFaultOut S= rtResetandOK.Q OR i_xVeto;
q_xFastFaultOut R= (NOT xOK OR xFastFaultRegFail) AND NOT i_xVeto;

//Reset OK for next cycle
xOK := True;

////////////////////////////////////////////////////////////////
END_ACTION

METHOD EvaluateOverrides : BOOL
VAR_INPUT
END_VAR
VAR
    FF : REFERENCE TO ST_FF;
    EvalIdx: DINT := 1;
END_VAR

FOR EvalIdx := 1 TO FF_ARRAY_UPPER_BOUND DO
    
    FF REF= astFF[EvalIdx];
    
    IF NOT FF.Info.InUse THEN 
        CONTINUE;
    ELSE
        // Veto timer
        IF FF.Ovrd.Deactivate THEN 
            FF.Ovrd.Timer.PT := T#0s; // Only needs to be set zero for one cycle
        ELSE
            FF.Ovrd.Timer.PT := UDINT_TO_TIME(FF.Ovrd.Duration);
        END_IF
        
        // UDINT conversions for ESS module compatibility.
        FF.Ovrd.Timer(
            IN := FF.Ovrd.Activate, // Rising edge activated
            Q => FF.Ovrd.Active);
            
        FF.Ovrd.tOvrdActivate(CLK:=FF.Ovrd.Active);
        FF.Ovrd.OvrdActLogAck S= FF.Ovrd.tOvrdActivate.Q;
        
        FF.Ovrd.tOvrdExpiring(CLK:=FF.Ovrd.Active);
        FF.Ovrd.OvrdExpLogAck S= FF.Ovrd.tOvrdExpiring.Q;
            
        FF.Ovrd.ElapsedTime := TIME_TO_UDINT(FF.Ovrd.Timer.ET);
        
        // Clear pushbuttons
        FF.Ovrd.Activate := FALSE;
        FF.Ovrd.Deactivate := FALSE;
        
    END_IF    
END_FOR
END_METHOD

{attribute 'obsolete' := 'Use EvaluateOverrides instead.'} 
METHOD EvaluateVetos : BOOL
VAR_INPUT
END_VAR
END_METHOD

METHOD ExecuteLogging : BOOL
VAR_INPUT
END_VAR
VAR
    FF : REFERENCE TO ST_FF;
    logIdx : DINT := 1; 
END_VAR

FOR logIdx := 1 to FF_ARRAY_UPPER_BOUND do
    
    FF REF= astFF[logIdx];
    
    IF NOT FF.Info.InUse THEN 
        CONTINUE;
    ELSE
        IF FF.FaultAck THEN
            
            pmpsTypeCode := 1;
            FormulateLogJson(FF);
            
            //Json is gen. in FormulateLogJson
            fbLogger(sMsg := 'Fast Fault, beam off', eSevr:=TcEventSeverity.Critical);
            
            FF.FaultAck := FALSE;
        END_IF
        
        IF FF.Ovrd.OvrdActLogAck THEN
            
            pmpsTypeCode := 2;
            FormulateLogJson(FF);
            
            fbLogger(sMsg := 'Veto activated', eSevr:=TcEventSeverity.Warning);
            
            FF.Ovrd.OvrdActLogAck := FALSE;
        END_IF
        
        IF FF.Ovrd.OvrdExpLogAck THEN
            
            pmpsTypeCode := 3;
            FormulateLogJson(FF);
            
            fbLogger(sMsg := 'Veto released', eSevr:=TcEventSeverity.Warning);
            
            FF.Ovrd.OvrdExpLogAck := FALSE;
        END_IF
    END_IF
END_FOR

// Log registration fault cleared
tFFRegFail(CLK:=xFastFaultRegFail);
IF tFFRegFail.Q THEN
    fbJson.StartObject();
    fbJson.AddKey('pmps_typecode');
    fbJson.AddUdint(5);
    fbJson.AddKey('pmps_path');
    fbJson.AddString(sPath);
    fbJson.EndObject();
    fbJson.CopyDocument(pDoc:=fbLogger.sJson, SIZEOF(fbLogger.sJson));
    fbLogger(sMsg := 'Fast fault registration failure cleared. This may be bad as a fast fault could go unoticed.', 
        eSevr:=TcEventSeverity.Warning);  
END_IF
END_METHOD

METHOD FormulateLogJson : STRING
VAR_INPUT
    FF : ST_FF;
END_VAR
fbJson.StartObject();
fbJson.AddKey('pmps_typecode');
fbJson.AddUdint(pmpsTypeCode);
fbJson.AddKey('pmps_path');
fbJson.AddString(FF.Info.sPath);
fbJson.AddKey('pmps_device_name');
fbJson.AddString(FF.Info.DevName);
fbJson.EndObject();
fbLogger.sJson := fbJson.GetDocument();
fbJson.ResetDocument();
END_METHOD

METHOD IdxCheckIn : BOOL
VAR_INPUT
    Idx : DINT;
    OK : BOOL;
    Reset : BOOL;
END_VAR
VAR
    stFF : ST_FF;
END_VAR
Idx := LIMIT(1,Idx,FF_ARRAY_UPPER_BOUND);
stFF := THIS^.astFF[Idx];

// Setting the log flag only on a state change.
stFF.FaultAck S= stFF.OK AND NOT OK;

// Updating internal fault state
stFF.OK := OK;

// Reset and latching logic
stFF.rtReset(CLK:=stFF.Reset OR Reset);
stFF.Reset R= stFF.rtReset.Q;
stFF.bsFF(SET := stFF.rtReset.Q OR stFF.Info.AutoReset, RESET1:= NOT OK);    

stFF.BeamPermitted := stFF.bsFF.Q1 OR stFF.Ovrd.Active;

// Fault generation    
IF NOT stFF.BeamPermitted THEN
    THIS^.xOK := FALSE; //Very clever, thanks Zach!
END_IF

// Fast fault accumulation
stFF.ftCountFault(CLK:=stFF.bsFF.Q1);
IF stFF.ftCountFault.Q THEN PMPS_GVL.AccumulatedFF := PMPS_GVL.AccumulatedFF + 1; END_IF

//Clear pushbuttons
stFF.Reset := FALSE;

// Copy state back to ff struct
THIS^.astFF[Idx] := stFF;
END_METHOD

METHOD Register : BOOL
VAR_INPUT
    stFFInfo : ST_FFInfo := (
        sPath := '',
        Desc := '',
        TypeCode := 16#00,
        DevName := ''); // Fast fault information
        
END_VAR
VAR_OUTPUT
    FFOName : T_MaxString;
    Idx : UINT;
END_VAR
VAR
END_VAR
FFOName := THIS^.sPath;
Idx := THIS^.nIndex;

IF THIS^.nIndex <= FF_ARRAY_UPPER_BOUND THEN
    
    THIS^.astFF[MIN(THIS^.nIndex,FF_ARRAY_UPPER_BOUND)].Info:=stFFInfo;
    
    THIS^.nIndex := THIS^.nIndex + 1;
    
    Register := TRUE; // Add successful    
ELSE
    fbJson.StartObject();
    fbJson.AddKey('pmps_typecode');
    fbJson.AddUdint(4);
    fbJson.AddKey('pmps_path');
    fbJson.AddString(stFFInfo.sPath);
    fbJson.AddKey('pmps_device_name');
    fbJson.AddString(stFFInfo.DevName);
    fbJson.EndObject();
    fbLogger.sJson := fbJson.GetDocument();
    fbJson.ResetDocument();
    fbLogger(sMsg:='Fast fault registration failed.',
        eSevr:=TcEventSeverity.Warning,
        eSubsystem:=E_Subsystem.MPS);
    xFastFaultRegFail := TRUE;
    Register := FALSE; // Failed to add name to list
END_IF
END_METHOD

END_FUNCTION_BLOCK

// ---- TestComponents/FB_Arbiter_Test.TcPOU
{attribute 'call_after_init'}
FUNCTION_BLOCK FB_Arbiter_Test EXTENDS TcUnit.FB_TestSuite
VAR_INPUT
END_VAR
VAR_OUTPUT
END_VAR
VAR
END_VAR

Arbitration();
RequestCheckRemoveBP();
FullArbitrationStack();

METHOD Arbitration
VAR_INPUT
END_VAR
VAR
    
     nAttReqID    :    UDINT    := 1;
    stAttReqBP    :    ST_BeamParams := PMPS_GVL.cstFullBeam;
    
    nPPEReqID    :    UDINT    := 2;
    stPPEReqBP    :    ST_BeamParams := PMPS_GVL.cstFullBeam;
    
    nEVReqID    :    UDINT    := 3;
    stEVReqBP    :    ST_BeamParams := PMPS_GVL.cstFullBeam;
    
    nRateReqID    :    UDINT    := 4;
    stRateReqBP    :    ST_BeamParams := PMPS_GVL.cstFullBeam;
    
    stArbitratedBP    :    ST_BeamParams;
    stExpectedBP    :    ST_BeamParams;
END_VAR
VAR_INST
    fbArbiter    :    FB_Arbiter(1);
END_VAR
TEST('Arbitration');

stAttReqBP.fAtt := 50;
stPPEReqBP.fPP_mJ := 1;
stEVReqBP.neVRange := 2#1111_1100_1111_1111;
stRateReqBP.nRate := 120;

//Load arbiter with beam parameter sets
AssertTrue(fbArbiter.AddRequest(nAttReqID, stAttReqBP),
                    'Safest attenuation request failed to load');
                    
//Load arbiter with beam parameter sets
AssertTrue(fbArbiter.AddRequest(nPPEReqID, stPPEReqBP),
                    'Safest PPE request failed to load');
                    
//Load arbiter with beam parameter sets
AssertTrue(fbArbiter.AddRequest(nEVReqID, stEVReqBP),
                    'Safest stEVReqBP request failed to load');
                    
//Load arbiter with beam parameter sets
AssertTrue(fbArbiter.AddRequest(nRateReqID, stRateReqBP),
                    'Safest stEVReqBP request failed to load');

stExpectedBP.fAtt     :=     stAttReqBP.fAtt;
stExpectedBP.fPP_mJ    :=  stPPEReqBP.fPP_mJ;
stExpectedBP.neVRange := stEVReqBP.neVRange;
stExpectedBP.nRate := stRateReqBP.nRate;

stArbitratedBP := fbArbiter.GetArbitratedBP();

AssertFalse(F_DifferentBeamParams(stExpectedBP, stArbitratedBP),
                'Arbitrated BP does not match expected.');

TEST_FINISHED();
END_METHOD

METHOD FullArbitrationStack
VAR_INPUT
END_VAR
VAR   
    nId    :    DWORD := 1;
    stReq    :    ST_BeamParams := (fAtt:=12);
END_VAR
VAR_INST
    fbArbiter    :    FB_Arbiter(1);
    
    fbHigherArb : FB_Arbiter(2);
    
    fbSubSysToArb : FB_SubSysToArbiter_IO; // Subsystem interface with beamline arbiter PLC
    pBPR : POINTER TO ST_BeamParams_IO;
    
    fbArbToSubSys : FB_ArbiterToSubSys_IO := (RequestingSystemID:=42); // Beamline arbiter PLC interface with subsystems
    pBPC : POINTER TO ST_BeamParams_IO;
    
    fbBPR : FB_BPRequestor; // Use in the arbiter PLC to apply an arbitrated beam parameter set to the accelerator interface
    
    FFO : FB_HardwareFFOutput; // Dummy FFO not important for these tests

    Cycle : INT := 0;
    
    CycleLimit : INT := 20;
    
END_VAR
VAR CONSTANT
    SysID : DWORD := 42;
END_VAR
// This simulates a synchronous cycle between the subsystem and arbiter PLC cycles. Ie. phase is locked, and cycle time is the same. This is not always the case, so these tests should be 
// trusted with a grain of salt.

TEST('FullStack');



CASE Cycle OF

0: 
    IF NOT fbArbiter.CheckRequestInPool(nID) THEN
        AssertTrue(fbArbiter.AddRequest(nId, stReq), 'Arbiter returned false from AddRequest'); // some device asking its local arbiter for some beam parameters
    END_IF  
    
    TEST('JustEnteredRequest');
    AssertFalse(fbArbiter.CheckRequest(nId),
        'Check should fail. Request not arbitrated yet.');
    TEST_FINISHED();
   
8000:
    TEST_FINISHED_NAMED('FullStack');   
    
END_CASE 


TEST('VerifyBPRHasBP');
IF fbHigherArb.CheckRequest(SysID) THEN
    AssertFalse(F_DifferentBeamParams(stReq, fbBPR.ReqBP),
        'Beam parameters not fully propagated to BPR at highest level');
        TEST_FINISHED_NAMED('VerifyBPRHasBP');
END_IF

TEST('ArbToSubsysPropagation');
IF fbArbToSubSys.nActiveCohort = fbArbToSubSys.nRequestedCohort THEN
    AssertTrue(fbHigherArb.CheckRequest(SysID),
        'Active cohort = Requested cohort before higher arbiter confirmed request was active');
    TEST_FINISHED_NAMED('ArbToSubsysPropagation');
END_IF

TEST('SubsysToArbPropagation');
IF fbArbiter.CheckRequest(nId) THEN
    AssertTrue(fbSubSysToArb.nActiveCohort >= fbSubSysToArb.nRequestCohort,
        'Request validated before higher level confirmation');
    TEST_FINISHED_NAMED('SubsysToArbPropagation');
END_IF


TEST('VerifyIncludedAtAllLevels');
IF fbArbiter.CheckRequest(nId) THEN
    AssertTrue(fbHigherArb.xActiveInArbitration, 'HigherArb is not yet included in arbitration');
    AssertTrue(fbArbiter.xActiveInArbitration, 'Local Arb is not yet included in arbitration');
    TEST_FINISHED_NAMED('VerifyIncludedAtAllLevels');
END_IF
      
    
///////////////////////////////////////
//Sub system cycle
fbSubSysToArb(Arbiter := fbArbiter, fbFFHWO := FFO);
//END of sub system cycle
///////////////////////////////////////

//Ethercat transfer simulation
// Transfer of requested BP to arbiter PLC
pBPR := ADR(fbArbToSubSys.i_RequestedBP);
pBPR^ := fbSubSysToArb.q_stRequestedBP;

// Transfer of current BP to sub system PLC
pBPC := ADR(fbSubSysToArb.i_stCurrentBP);
pBPC^ := fbArbToSubSys.o_CurrentBP;

//////////////////////////////////////
//Start of arbiter plc cycle
//Arb io collects sub system status
fbArbToSubSys(Arbiter := fbHigherArb, fbFFHWO := FFO); // This is making a request in the higher arb
//BPR collects arbiter summation
fbBPR(Arbiter := fbHigherArb); // This is getting the arbitrated BP




IF CycleLimit > Cycle THEN
    Cycle := Cycle + 1;
ELSE 
    Cycle := 8000;
END_IF
END_METHOD

METHOD RequestCheckRemoveBP
VAR_INPUT
END_VAR
VAR
    
    nId    :    DWORD := 1;
    stReq    :    ST_BeamParams;
END_VAR
VAR_INST
    fbArbiter    :    FB_Arbiter(1);
END_VAR
TEST('RequestBP');
AssertTrue(fbArbiter.AddRequest(nId, stReq),
    'Request failed');

TEST_FINISHED();
    
TEST('DuplicateID');
AssertFalse(fbArbiter.AddRequest(nId, stReq),
    'Duplicate request accepted, not good.');

TEST_FINISHED();
    
TEST('CheckBP');
AssertFalse(fbArbiter.CheckRequest(nId),
    'Check should fail. Request not arbitrated yet.');
TEST_FINISHED();

TEST('CheckBPArbitrated');
WRITE_PROTECTED_ULINT(ADR(fbArbiter.nArbiterCohort), fbArbiter.nArbiterCohort + 1);
AssertTrue(fbArbiter.CheckRequest(nId),
    'Check should pass.');

TEST_FINISHED();      
    
TEST('IDDoesNotExist');
WRITE_PROTECTED_ULINT(ADR(fbArbiter.nArbiterCohort), fbArbiter.nArbiterCohort + 1); 
AssertFalse(fbArbiter.CheckRequest(nId+1),
    'Check returned true when ID does not exist');

TEST_FINISHED();
    
TEST('RemoveBP');
AssertTrue(fbArbiter.RemoveRequest(nId),
    'Remove failed');
AssertFalse(fbArbiter.CheckRequest(nId),
    'Remove did not remove request');
    
TEST_FINISHED();
END_METHOD

END_FUNCTION_BLOCK

// ---- MajorComponents/InterPlcComm/FB_SubSysToArbiter_IO.TcPOU
// Use on a subsystem PLC to request from the arbiter
// Run at the top of your cycle to receive the latest BP
FUNCTION_BLOCK FB_SubSysToArbiter_IO IMPLEMENTS I_HigherAuthority
VAR_INPUT
    Reset : BOOL; // Fast fault reset
END_VAR
VAR_OUTPUT
END_VAR
VAR_IN_OUT
	Arbiter	: FB_Arbiter;
    fbFFHWO : FB_HardwareFFOutput;
END_VAR
VAR
    {attribute 'TcLinkTo' := 'TIIB[PMPS_PRE]^IO Inputs^CurrentBP'}
    i_stCurrentBP    AT %I* :    ST_BeamParams_IO;
    {attribute 'TcLinkTo' := 'TIIB[PMPS_PRE]^IO Outputs^RequestedBP'}
    q_stRequestedBP AT %Q* :    ST_BeamParams_IO;
    {attribute 'pytmc' := 'pv: TxPDO_toggle
        io: i'}
    {attribute 'TcLinkTo' := 'TIIB[PMPS_PRE]^SYNC Inputs^TxPDO toggle'}
    xTxPDO_toggle    AT     %I* :    BIT;
    {attribute 'pytmc' := 'pv: TxPDO_state
        io: i'}
    {attribute 'TcLinkTo' := 'TIIB[PMPS_PRE]^SYNC Inputs^TxPDO state'}
    xTxPDO_state    AT    %I*    :    BIT;
    
    
    // Fast faults
    ffPMPSIO_Disconnect : FB_FastFault := (i_Desc:='Arbiter network interface disconnected or not OP');
    
    // A request is not considered included until the active cohort number is >= the request cohort number.
    {attribute 'pytmc' := 'pv: RequestCohort
        io: i'}
    nRequestCohort : UDINT := 0; // Request cohort
    {attribute 'pytmc' := 'pv: ActiveCohort
        io: i'}
    nActiveCohort : UDINT := 0; // Active cohort, updated by incoming BP from arbiter PLC, in the ElevateRequest arbiter call

END_VAR

//Receiving current BP state
PMPS_GVL.stCurrentBeamParameters := IO_TO_BP(i_stCurrentBP);
PMPS_GVL.stCurrentBeamParameters.xValidToggle := xTxPDO_state; // This line must follow the one above. Sequence is important.

// Forwarding BP request for the subsystem
Arbiter.ElevateRequest(THIS^);

//Broadcasting current request
PMPS_GVL.stRequestedBeamParameters := IO_TO_BP(q_stRequestedBP);


q_stRequestedBP.xValid := TRUE; // This is set and held true here every cycle to prove the PLC on this side is still running

ffPMPSIO_Disconnect(io_fbFFHWO := fbFFHWO,
    i_xReset := Reset);

METHOD CheckRequest : BOOL
VAR_INPUT
	nReqID	: DWORD;
END_VAR
VAR_INST
    xFirstTime : BOOL := TRUE;
    nId : DWORD;
END_VAR
// Check this id matches what we've seen before
IF xFirstTime THEN
    nId := nReqId;
ELSIF nId <> nReqId THEN
    PMPS_GVL.fbLog(sMsg := 'SubSysToArbiter Check mismatched with a different ID', eSevr := TcEventSeverity.Error);
    RETURN;
END_IF

nActiveCohort := ULINT_TO_UDINT(i_stCurrentBP.nCohortInt);

// i_stCurrentBP.nCohortInt is incremented by the FB_ArbiterToSubSys block on the other side of the EL669* interface
CheckRequest := nRequestCohort <= nActiveCohort;
END_METHOD

METHOD RequestBP : BOOL
VAR_INPUT
	(*StateID of state requesting beam parameter set*)
	nReqID	: DWORD;
	(*Requested beam params*)
	stReqBP	: ST_BeamParams;
END_VAR
// Check the request is coming from the same source we're used to

// Update internal BP request struct
q_stRequestedBP := BP_TO_IO(stReqBP);

nRequestCohort := nRequestCohort + 1;

// Mark the current cohort id
q_stRequestedBP.nCohortInt := nRequestCohort;

RequestBP := TRUE;
END_METHOD

END_FUNCTION_BLOCK

// ---- MajorComponents/InterPlcComm/FB_ArbiterToSubSys_IO.TcPOU
(* Exchanges preemption requests and current beam state with subsystems in arbiter
network.

2019-12-2, A. Wallace

*)
FUNCTION_BLOCK FB_ArbiterToSubSys_IO
VAR_INPUT
	RequestingSystemID	:	DWORD := PMPS_GVL.EXCLUDED_ASSERTION_ID; // System ID for making requests to the supreme arbiter
    Reset : BOOL;
END_VAR
VAR_OUTPUT
END_VAR
VAR_IN_OUT
	Arbiter	: FB_Arbiter;
    fbFFHWO : FB_HardwareFFOutput;
END_VAR
VAR
    
	i_RequestedBP AT %I*	:	ST_BeamParams_IO; // Requested BP from subsystem
    {attribute 'pytmc' := '
        pv: RequestedBP:FromSubSys
    '}
    RequestedBP: ST_BeamParams;
    
	o_CurrentBP AT %Q* : ST_BeamParams_IO; // Current BP set
    
    // EL6692 Diagnostics
    i_Connected AT %I* : BOOL; // SYNC Inputs^External device not connected !!! Doesn't really work.
    {attribute 'pytmc' := 'pv: WcState
        io: i
        field: DESC Working counter state.
        field: ZNAM OK
        field: ONAM Error'}
    i_WcState AT %I* : BOOL; // WcState^WcState
    {attribute 'pytmc' := 'pv: TxPDO_state
        io: i
        field: DESC PDO Transmission is OK
        field: ZNAM OK
        field: ONAM Error'}
    i_TxPDOState AT %I* : BOOL; // SYNC Inputs^TxPDO state
    {attribute 'pytmc' := 'pv: TxPDO_toggle
        io: i
        field: DESC PDO Transmission is OK
        field: ZNAM OK
        field: ONAM Error'}
    i_TxPDOToggle AT %I* : BOOL; // TxPDO toggle
    
    // Fast faults
    ffPMPSIO_Disconnect : FB_FastFault := (i_Desc:='Fast fault on arbiter disconnection'); // Fast fault for ethercat issues
    nActiveCohort : UDINT := 0; // Active cohort. Updated to the req. number from the sub system after request is confirmed.
    nRequestedCohort : UDINT := 0;
    rtToggle : R_TRIG;

	
END_VAR


RequestedBP := IO_TO_BP(i_RequestedBP);

// Update arbiter with our request
rtToggle(CLK:= i_RequestedBP.xValid); // If interface resumes, reset/catch up
// xValid will go false if the PLC program on the other side is stopped. Ironically the ethercat interface continues happily.
IF i_RequestedBP.nCohortInt > nRequestedCohort OR rtToggle.Q THEN // If subsystem cohort has incremented, update beam parameter request with our arbiter
    Arbiter.RemoveRequest(RequestingSystemID);
    Arbiter.AddRequest(RequestingSystemID, RequestedBP);
    nRequestedCohort := i_RequestedBP.nCohortInt;
END_IF


// Check if latest request is acknowledged by this arbiter
// This happens after an arbitration
IF Arbiter.CheckRequest(RequestingSystemID) THEN
    nActiveCohort := nRequestedCohort; // If it is, then the active cohort is set to the requested cohort number.
END_IF

// Sending current beam parameter set to subsystems 
o_CurrentBP := BP_TO_IO(PMPS_GVL.stCurrentBeamParameters);
o_CurrentBP.nCohortInt := nActiveCohort;


//////////////////////////////////////
// Verifying the ethercat interface health
/////////////////////////////////////
// Both of these values should be 0 for a fully valid exchange
ffPMPSIO_Disconnect.i_xOK := NOT i_WcState AND NOT i_TxPDOState;

ffPMPSIO_Disconnect(
    io_fbFFHWO := fbFFHWO,
    i_xReset := Reset);

END_FUNCTION_BLOCK

// ---- MajorComponents/FB_BPRequestor.TcPOU
(* BP Requestor
Elevates the BP request from an arbiter to PMPS_GVL.stRequestedBP
*)
FUNCTION_BLOCK FB_BPRequestor IMPLEMENTS I_HigherAuthority
VAR_INPUT
END_VAR
VAR_OUTPUT
    q_ReqBP : ST_BeamParams; // Arbitrated BP
END_VAR
VAR_IN_OUT
    Arbiter : FB_Arbiter;
    //FFO : FB_HardwareFFOutput;
END_VAR
VAR
    ReqBP : ST_BeamParams;
    nCohort : ULINT; // Current cohort, inc. 1 cycle after IO is updated
    nRequestCohort : ULINT; // Cohort number recorded at the time of the request.
END_VAR

Arbiter.ElevateRequest(THIS^); // Executes arbitration and retrieves ReqBP

IF nRequestCohort >= nCohort THEN
    // Update requested BP set
    q_ReqBP := ReqBP;
    // Note: we may do more here someday... perhaps all of the output control
    // will reside in here, and be solely controlled by this block. For now
    // I am going to adopt a flat management structure.
    // Start a new cohort
    nCohort := nCohort + 1;
END_IF

// Returns true when outputs to MPS are updated
METHOD CheckRequest : BOOL
VAR_INPUT
	nReqID	: DWORD;
END_VAR
VAR_INST
    xFirstTime : BOOL;
    nId : DWORD;
END_VAR
(* nRequestCohort will be < nCohort after output control
function blocks have been updated to reflect the new request
*)
CheckRequest := nRequestCohort < nCohort;
END_METHOD

METHOD RequestBP : BOOL
VAR_INPUT
	(*StateID of state requesting beam parameter set*)
	nReqID	: DWORD;
	(*Requested beam params*)
	stReqBP	: ST_BeamParams;
END_VAR
VAR_INST
    ReqID : DWORD;
    Registered : BOOL := FALSE;
END_VAR

// Check the request is coming from the same source we're used to
IF NOT Registered THEN
    ReqID := nReqID;
    Registered := TRUE;
END_IF
// log a complaint if false
RequestBP := ReqId = nReqId;

// Update internal BP request struct
ReqBP := stReqBP;

// Record current cohort
IF nRequestCohort = 0 THEN
    nRequestCohort := 1;
ELSE
    nRequestCohort := nCohort;
END_IF
END_METHOD

END_FUNCTION_BLOCK

// ---- TestComponents/FB_SubsysToArb_Test.TcPOU
{attribute 'call_after_init'}
FUNCTION_BLOCK FB_SubsysToArb_Test EXTENDS TcUnit.FB_TestSuite
VAR_INPUT
END_VAR
VAR_OUTPUT
END_VAR
VAR
END_VAR

BasicFunction();

METHOD BasicFunction
VAR_INPUT
END_VAR
VAR   
    nId    :    DWORD := 1;
    stReq    :    ST_BeamParams := (fAtt:=12);
END_VAR
VAR_INST
    fbArbiter    :    FB_Arbiter(1);
    
    fbSubSysToArb : FB_SubSysToArbiter_IO; // Subsystem interface with beamline arbiter PLC
    pBPC : POINTER TO ST_BeamParams_IO;
    
    ioCurrentBP : ST_BeamParams_IO; 
    
    FFO : FB_HardwareFFOutput; // Dummy FFO not important for these tests
    
END_VAR
VAR CONSTANT
    SysID : DWORD := 42;
END_VAR
// This simulates a synchronous cycle between the subsystem and arbiter PLC cycles. Ie. phase is locked, and cycle time is the same. This is not always the case, so these tests should be 
// trusted with a grain of salt.

TEST('Add to arbiter');

IF NOT fbArbiter.CheckRequestInPool(nID) THEN
    AssertTrue(fbArbiter.AddRequest(nId, stReq), 'Arbiter returned false from AddRequest'); // some device asking its local arbiter for some beam parameters
END_IF  
   
TEST_FINISHED();   

///////////////////////////////////////
//Sub system cycle
fbSubSysToArb(Arbiter := fbArbiter, fbFFHWO := FFO);
//END of sub system cycle
///////////////////////////////////////


TEST('Initial Elevation');
AssertTrue(fbSubSysToArb.nRequestCohort = fbSubSysToArb.q_stRequestedBP.nCohortInt, 'ReqCohort and qBP Cohort do not match');
AssertFalse(fbArbiter.xActiveInArbitration, 'Arbiter indicates it is included in arbitration prematurely');
AssertTrue(fbSubSysToArb.nRequestCohort = 1, 'Cohort index should move to 1 with first request');
TEST_FINISHED_NAMED('Initial Elevation');
    
//Ethercat transfer simulation
// Transfer of requested BP to arbiter PLC
// pBPR := ADR(fbArbToSubSys.i_RequestedBP);
// pBPR^ := fbSubSysToArb.q_stRequestedBP;

ioCurrentBP := fbSubSysToArb.q_stRequestedBP;
// NOTE: Setting the returning cohort number to something less than the request cohort number
// will prevent the sub system arbiter FB from considering itself active in arbitration.
// The next set of tests verify this.
ioCurrentBP.nCohortInt := 0;

// Transfer of current BP to sub system PLC
pBPC := ADR(fbSubSysToArb.i_stCurrentBP);
pBPC^ := ioCurrentBP;

///////////////////////////////////////
//Sub system cycle
fbSubSysToArb(Arbiter := fbArbiter, fbFFHWO := FFO);
//END of sub system cycle
///////////////////////////////////////

TEST('Not yet active in arbitration');
AssertTrue(fbSubSysToArb.nActiveCohort = 0, 'Active cohort should still be zero, per ioCurrentBP.nCohortInt setting above.');
AssertFalse(fbArbiter.xActiveInArbitration, 'Arbiter indicates it is included in arbitration prematurely, checkrequest might be broken');
AssertTrue(fbSubSysToArb.nRequestCohort = 1, 'Cohort index should remain at 1 because there have been no additional requests added to the arbiter');
TEST_FINISHED_NAMED('Not yet active in arbitration');

//Ethercat transfer simulation
// Transfer of requested BP to arbiter PLC
// pBPR := ADR(fbArbToSubSys.i_RequestedBP);
// pBPR^ := fbSubSysToArb.q_stRequestedBP;

ioCurrentBP := fbSubSysToArb.q_stRequestedBP;
// NOTE: Now we simulate the FB_ArbiterToSubSys_IO updating the cohort number to the same value as the request cohort, indicating that cohort has been included
ioCurrentBP.nCohortInt := 1;

// Transfer of current BP to sub system PLC
pBPC := ADR(fbSubSysToArb.i_stCurrentBP);
pBPC^ := ioCurrentBP;

///////////////////////////////////////
//Sub system cycle
fbSubSysToArb(Arbiter := fbArbiter, fbFFHWO := FFO);
//END of sub system cycle
///////////////////////////////////////

TEST('Active in arbitration');
AssertTrue(fbSubSysToArb.nActiveCohort = fbSubSysToArb.nRequestCohort, 'Active cohort and request cohort do not match');
AssertTrue(fbArbiter.xActiveInArbitration, 'Arbiter does not indicate it is included in higher arbitration');
TEST_FINISHED_NAMED('Active in arbitration');
END_METHOD

END_FUNCTION_BLOCK

// ---- TestComponents/FB_ArbToSubsys_Test.TcPOU
{attribute 'call_after_init'}
FUNCTION_BLOCK FB_ArbToSubsys_Test EXTENDS TcUnit.FB_TestSuite
VAR_INPUT
END_VAR
VAR_OUTPUT
END_VAR
VAR
END_VAR

BasicFunction();

METHOD BasicFunction
VAR_INPUT
END_VAR
VAR CONSTANT
    SysID : DWORD := 42;
END_VAR
VAR   
    nId    :    DWORD := 1;
    stReq    :    ST_BeamParams := (fAtt:=12);
END_VAR
VAR_INST
    fbArbiter    :    FB_Arbiter(1);
    
    pBPR : POINTER TO ST_BeamParams_IO;
    
    stBPRIO : ST_BeamParams_IO := (
        nCohortInt := 1,
        fAtt := 35); // Simulates subsystem BP request
    
    fbArbToSubSys : FB_ArbiterToSubSys_IO := (RequestingSystemID:=42); // Beamline arbiter PLC interface with subsystems
    pBPC : POINTER TO ST_BeamParams_IO;
    
    fbBPR : FB_BPRequestor; // Use in the arbiter PLC to apply an arbitrated beam parameter set to the accelerator interface
    
    FFO : FB_HardwareFFOutput; // Dummy FFO not important for these tests

    Cycle : INT := 0;
    
    CycleLimit : INT := 20;
    
END_VAR

// Simulate an initial cycle with no new requests coming in
fbArbToSubSys(Arbiter:=fbArbiter, fbFFHWO:=FFO);

TEST('Init');
TEST_FINISHED();

//Ethercat transfer simulation
// Transfer of requested BP to arbiter PLC
pBPR := ADR(fbArbToSubSys.i_RequestedBP);
pBPR^ := stBPRIO;

///////////////////////////////////////
//Sub system cycle
fbArbToSubSys(Arbiter:=fbArbiter, fbFFHWO:=FFO);
//END of sub system cycle
///////////////////////////////////////


TEST('New request');
    AssertTrue(fbArbToSubSys.nRequestedCohort = fbArbToSubSys.i_RequestedBP.nCohortInt, 'ReqCohort and qBP Cohort do not match, and they should');
    AssertTrue(fbArbiter.CheckRequestInPool(SysID), 'ArbToSubSys request should be in arbiter pool now');
    AssertTrue(fbArbToSubSys.nActiveCohort = 0, 'Active cohort should remain the initial value until the current request is active in higher arbitration');
    AssertTrue(fbArbToSubSys.o_CurrentBP.nCohortInt = fbArbToSubSys.nActiveCohort, 'Cohort being sent to sub system remains unincremented');
TEST_FINISHED_NAMED('New request');
    

///////////////////////////////////////
//Sub system cycle
fbBPR(Arbiter:=fbArbiter);
fbArbToSubSys(Arbiter:=fbArbiter, fbFFHWO:=FFO);
//END of sub system cycle
///////////////////////////////////////

///////////////////////////////////////
//Sub system cycle
fbBPR(Arbiter:=fbArbiter);
fbArbToSubSys(Arbiter:=fbArbiter, fbFFHWO:=FFO);
//END of sub system cycle
///////////////////////////////////////


TEST('Request has become active');
    AssertTrue(fbArbToSubSys.nRequestedCohort = fbArbToSubSys.nActiveCohort, 'ReqCohort and qBP Cohort do not match, and they should');
    AssertTrue(fbArbiter.CheckRequest(SysID), 'ArbToSubSys request should be in arbiter pool now');
    AssertTrue(fbArbToSubSys.nActiveCohort = stBPRIO.nCohortInt, 'Active cohort should remain the initial value until the current request is active in higher arbitration');
    AssertTrue(fbBPR.q_ReqBP.fAtt = stBPRIO.fAtt, 'BPR and requested BP should match');
TEST_FINISHED_NAMED('Request has become active');
END_METHOD

END_FUNCTION_BLOCK

// ---- MajorComponents/FastFaults/FB_FastFaultLogger.TcPOU
FUNCTION_BLOCK FB_FastFaultLogger
VAR_INPUT
END_VAR
VAR_OUTPUT
END_VAR
VAR
END_VAR

END_FUNCTION_BLOCK

// ---- MajorComponents/FB_LinearDeviceStateTable.TcPOU
(* This function block implements simple database. Data element values are stored in the hash table.  *)
FUNCTION_BLOCK FB_LinearDeviceStateTable
VAR_INPUT
    key         : DWORD := 0;(* Entry key: used by A_Lookup, A_Remove method, the key variable is also used by A_Add method *)
    putPosPtr    : POINTER TO T_HashTableEntry := 0;(* Hash table entry position pointer (used by A_Find, A_GetNext, A_GetPrev) *)
    putValue     : ST_DeviceState;(* Hash table entry value (used by A_AddHead, A_AddTail, A_Find )*)
END_VAR
VAR_OUTPUT
    bOk            : BOOL := FALSE;(* TRUE = Success, FALSE = Failed *)
    getPosPtr    : POINTER TO T_HashTableEntry := 0;(* Returned hash table entry position pointer *)
    getValue     : ST_DeviceState;(* Returned hash table entry value *)
    nCount        : UDINT := 0;(* Hash table size (number of used entries, used by A_Count) *)
END_VAR
VAR
    dataPool    : ARRAY[0..PMPS_GVL.MAX_DEVICE_STATES] OF ST_DeviceState;(* Structured data element pool *)
    entries        : ARRAY[0..PMPS_GVL.MAX_DEVICE_STATES] OF T_HashTableEntry;(* Max. number of hash table entries. The value of table entry = 32 bit integer (pointer to dataPool-array-entry) *)
    fbTable     : FB_HashTableCtrl;(* basic hash table control function block *)
    hTable         : T_HHASHTABLE;(* hash table handle *)
    pRefPtr        : POINTER TO ST_DeviceState := 0;
    indexOfElem    : ULINT;(* Integer value (max. size: x86=>32bit, x64=>64bit)*)
END_VAR

;

ACTION A_Add:
(* Adds entry to the table *)
MEMSET( ADR( getValue ), 0, SIZEOF( getValue ) );
getPosPtr := 0;

fbTable.A_Add( hTable := hTable, key := key, putValue := ADR(PMPS_GVL.cstSafeBeam)(* we will set this value later *), getPosPtr=>getPosPtr, bOk=>bOk );(* Add new element to the table, getPosPtr points to the new entry *)
IF fbTable.bOk THEN(* Success *)
    fbTable.A_GetIndexAtPosPtr( hTable := hTable, putPosPtr := getPosPtr, getValue =>indexOfElem, bOk=>bOk );(* Get array index of getPosPtr entry *)
    IF fbTable.bOk THEN(* Success *)
        pRefPtr     := ADR( dataPool[indexOfElem] );(* Get pointer to the data element *)

        pRefPtr^ := putValue;(* copy application value *)

        fbTable.A_Add( hTable := hTable, key := key, putValue := pRefPtr, bOk=>bOk );(* Assign the entry value = pointer to the data element *)
        IF fbTable.bOk THEN(* Success *)
            getValue := putValue;
        END_IF
    END_IF
END_IF
END_ACTION

ACTION A_Count:
(* Count number of used entries *)
nCount := hTable.nCount;
bOk := TRUE;
END_ACTION

ACTION A_GetFirst:
(* Get first entry position pointer and value *)
MEMSET( ADR( getValue ), 0, SIZEOF( getValue ) );
getPosPtr := 0;

fbTable.A_GetFirst( hTable := hTable, putPosPtr := putPosPtr, getValue=>pRefPtr, getPosPtr=>getPosPtr, bOk=>bOk );
IF fbTable.bOk THEN
    getValue := pRefPtr^;
END_IF
END_ACTION

ACTION A_GetNext:
(* Get next entry position pointer and value *)
MEMSET( ADR( getValue ), 0, SIZEOF( getValue ) );
getPosPtr := 0;
bOk := FALSE;

IF putPosPtr = 0 THEN
    RETURN;
END_IF

fbTable.A_GetNext( hTable := hTable, putPosPtr := putPosPtr, getValue=>pRefPtr, getPosPtr=>getPosPtr, bOk=>bOk );
IF fbTable.bOk THEN
    getValue := pRefPtr^;
END_IF
END_ACTION

ACTION A_Lookup:
(* Lookup for entry by key  *)
MEMSET( ADR( getValue ), 0, SIZEOF( getValue ) );
getPosPtr := 0;

fbTable.A_Lookup( key := key, hTable := hTable, putPosPtr := putPosPtr, getValue=>pRefPtr, getPosPtr=>getPosPtr, bOk=>bOk );
IF fbTable.bOk THEN
    getValue := pRefPtr^;
END_IF
END_ACTION

ACTION A_Remove:
(* Search for entry and remove it *)
MEMSET( ADR( getValue ), 0, SIZEOF( getValue ) );
getPosPtr := 0;

fbTable.A_Remove( key := key, hTable := hTable, putPosPtr := putPosPtr, getValue=>pRefPtr, getPosPtr=>getPosPtr, bOk=>bOk );
IF fbTable.bOk THEN
    getValue := pRefPtr^;
END_IF
END_ACTION

ACTION A_Reset:
(* Reset/initialize linked list *)
MEMSET( ADR( getValue ), 0, SIZEOF( getValue ) );
getPosPtr := 0;
bOk := F_CreateHashTableHnd( ADR( entries ), SIZEOF( entries ), hTable );(* Intialize table handle *)
fbTable.A_Reset( hTable := hTable, bOk=>bOk );
nCount := 0;
END_ACTION

END_FUNCTION_BLOCK

// ---- MajorComponents/FB_LinearGovernor.TcPOU

(* The governor is meant to check your work and keep you from making mistakes.

Checks:
Does your state match the device position and visa versa?
Are the beam parameters safe for the device state?
Did you properly assert the transition and final beam parameters?

*)
FUNCTION_BLOCK FB_LinearGovernor
VAR_INPUT
    i_stCurrentBeamParams    :    ST_BeamParams; //Link to global beam params
    i_xMPSOverride            :    BOOL; //True releases MPS limits after a delay
    i_xTransitionRequested    :    BOOL; //Set true to request a transition
    i_xResetMPSFault    :    BOOL; //Set true to clear MPS fault 
END_VAR
VAR_OUTPUT
     //True when governor has released restrictions
    q_xTransitionPermitted    :    BOOL;
    //Set if MC_Power has an error, or override mode is requested
    q_xFault    :    BOOL; 
    // Indicates override mode is active
    q_xMPSLimitsOverridden: BOOL;
END_VAR
VAR_IN_OUT
    stDevice    :    ST_Device; //The governed
    Arbiter    :    FB_Arbiter;
    FastFaultOutput    :    FB_HardwareFFOutput;
END_VAR
VAR
    mcPower    :    MC_Power;
    
    xActuatorPositiveEnable: BOOL;
    xActuatorNegativeEnable: BOOL;
    
    xMPSPositiveEnable    :    BOOL;
    xMPSNegativeEnable    :    BOOL;
    lrPosition: LREAL;
    
    lrLatchedTargetPosition    :    LREAL;
    lrLatchedTargetTolerance    :    LREAL;
    stLatchedTargetState    :    ST_DeviceStateExt;
    
    lrMPSUpperLimit: LREAL;
    lrMPSLowerLimit: LREAL;
    rtNewState: R_TRIG;
    xTransitionOK: BOOL;
    
    tonMPSOverrideMode    :    TON := (
        PT := T#5S
    );
    
    srMPSFault    :    SR;
    // Actuator out of bounds fault
    xActuatorOOB: BOOL;
    //Beam parameters out of spec
    xBeamParamsOOS: BOOL;
    //Beam parameters of currently latched state
    
    stLatchedBeamParams: ST_BeamParams;
    stTargetState: ST_DeviceStateExt;
    
    rtLatchNewState    :    R_TRIG;
    xInit: BOOL := TRUE;
    
    stInitDeviceState: ST_DeviceStateExt;
    // Indicates an error with initialization
    xInitFault: BOOL;
    // Indicates the state could not be found in the state table. There may be something wrong in the device state machine implementation or state table instantiation.
    xStateLookupError: BOOL;
    // A transition needs to be requested at least once before we start latching any state.
    xTransitionHasBeenRequested: BOOL := FALSE;
    ffBeamParamsOK : FB_FastFault;
    ffActuatorBoundsOK    :    FB_FastFault;
END_VAR


lrPosition := stDevice.stAxis.NcToPlc.ActPos; //Actuator position

stDevice.stAxis.ReadStatus();
//Init
(* The init strategy is:
If the device is restored and it's residing at the safe position,
no PMPS faults. *)
////////////////////////////////
    IF xInit THEN
        xInit := FALSE;
        //Use nSafeSate for initialization. 
        stDevice.StateTable.A_Lookup(key := stDevice.nSafeState);
        IF stDevice.StateTable.bOk THEN
            stInitDeviceState := F_DeviceState_To_DeviceStateExt(stDevice.StateTable.getValue, TRUE);
            xInitFault := FALSE;
        ELSE
            xInitFault := TRUE;
            stInitDeviceState.xValid := FALSE;
        END_IF
        lrLatchedTargetPosition := stInitDeviceState.rPosition;
        lrLatchedTargetTolerance := stInitDeviceState.rTolerance;
        stLatchedBeamParams := stInitDeviceState.stReqBeamParam;
    END_IF

// The governor will permit transitions once it verifies the transition assertion is active
// Note the governor does not verify the target state beam params are asserted, perhaps it should <TODO>
////////////////////////////////
    IF i_xTransitionRequested THEN
        xTransitionHasBeenRequested    := TRUE;
        
        xTransitionOK := Arbiter.CheckRequest( stDevice.stTransitionState.nStateRef) AND F_SafeBPCompare(i_stCurrentBeamParams, stDevice.stTransitionState.stReqBeamParam);
        
        //Set the target state for evaluation in further logic
        stdevice.StateTable.A_Lookup(key := stDevice.nTargetState);
        IF stDevice.StateTable.bOk THEN
            stTargetState := F_DeviceState_To_DeviceStateExt(stDevice.StateTable.getValue, TRUE);
            xStateLookupError := FALSE;
        ELSE
            xStateLookupError := TRUE;
            stTargetState.xValid := FALSE;
        END_IF
    ELSE
        xTransitionOK := FALSE;
    END_IF

(* Note about TransitionRequested

If TransitionRequested goes false during a transition, an MPS fault may be induced. This occurs
because the Actuator Out of Bounds fault will go back to using the original state limits, which
the axis may have already moved beyond.

To avoid this transient fault, make sure your device state machine is implemented such that the 
transition request to the governor block remains high until the target position is reached.
*)

//Determine if a transition is complete and latch the new state
(* A transition is complete when:

Axis at standstill.
Axis within tolerance.
No transition req.

Once these conditions are met, the MPS limits shall re-engage to restrict the
axis motion to the tolerance around the state position and the MPS fault monitors
shall evaluate based on the newly latched target state.
*)

rtLatchNewState(CLK := stDevice.stAxis.Status.StandStill AND
    lrPosition <= stTargetState.rPosition + stTargetState.rTolerance AND
    lrPosition >= stTargetState.rPosition - stTargetState.rTolerance AND
    NOT i_xTransitionRequested AND xTransitionHasBeenRequested);
    
IF rtLatchNewState.Q THEN
    lrLatchedTargetPosition := stTargetState.rPosition;
    lrLatchedTargetTolerance := stTargetState.rTolerance;
    stLatchedBeamParams := stTargetState.stReqBeamParam;
    stLatchedTargetState := stTargetState;
END_IF

//Let other blocks know the governor won't interfer with transitions
q_xTransitionPermitted := xTransitionOK;

//Adjust limit ranges based on active state and current target
IF xTransitionOK THEN
    //Extend range to include target state
    lrMPSUpperLimit := MAX(lrMPSUpperLimit, stTargetState.rPosition + stTargetState.rTolerance);
    lrMPSLowerLimit := MIN(lrMPSLowerLimit, stTargetState.rPosition - stTargetState.rTolerance);
ELSE
    //Calculate the limit positions for MPS based on current state
    lrMPSUpperLimit := lrLatchedTargetPosition + lrLatchedTargetTolerance;
    lrMPSLowerLimit := lrLatchedTargetPosition - lrLatchedTargetTolerance;
END_IF


//MPS override
(* In override mode, the device will be free to move anywhere within it's travel range *)
//Permit motion after a small delay
tonMPSOverrideMode(IN:=i_xMPSOverride OR stDevice.xOverrideMPSLimits, Q=>q_xMPSLimitsOverridden);

//Virtual limit switch evaluation
xActuatorPositiveEnable    := stDevice.i_xHiLim AND lrPosition <= stDevice.lrUpperPositionLimit;
xActuatorNegativeEnable    := stDevice.i_xLoLim AND lrPosition >= stDevice.lrLowerPositionLimit;

//Evaluate MPS limit states
xMPSPositiveEnable := lrPosition <= lrMPSUpperLimit;
xMPSNegativeEnable := lrPosition >= lrMPSLowerLimit;

//Final Limit switch evaluation
mcPower.Enable_Positive := xActuatorPositiveEnable AND (tonMPSOverrideMode.Q OR xMPSPositiveEnable);
mcPower.Enable_Negative := xActuatorNegativeEnable AND (tonMPSOverrideMode.Q OR xMPSNegativeEnable);

mcPower(
    Axis := stDevice.stAxis,
    Enable := stDevice.xEnable //link to device enable <TODO>
);



//MPS Faults
//Fault if the beam is unsafe for current state
ffBeamParamsOK(i_xOK:=F_SafeBPCompare(i_stCurrentBeamParams, stLatchedBeamParams), 
                i_xReset:=i_xResetMPSFault,
                io_fbFFHWO := FastFaultOutput);

//Fault if the position is outside of the permitted range
ffActuatorBoundsOK(i_xOK := (lrPosition <= lrMPSUpperLimit AND lrPosition >= lrMPSLowerLimit), 
                    i_xReset:=i_xResetMPSFault,
                io_fbFFHWO := FastFaultOutput);


    
//Collect all other faults
q_xFault := NOT ffBeamParamsOK.o_xFFLine OR
    NOT ffActuatorBoundsOK.o_xFFLine OR
    mcPower.Error    OR
    i_xMPSOverride    OR
    xInitFault;

//Any faults trip the fast fault line for this FB    
//FastFaultOutput.CheckIn(NOT q_xFault);

END_FUNCTION_BLOCK

// ---- MajorComponents/PMPS_MPS_Interface/FB_BeamClassOutputs.TcPOU
(*
Sets the beam class assertion lines for a given beam class.
*)
FUNCTION_BLOCK FB_BeamClassOutputs
VAR_INPUT
    BP : ST_BeamParams;
END_VAR
VAR_OUTPUT
END_VAR
VAR
    nBeamClass   :    BYTE;
    wBeamClass    :    BYTE;

    InitCounter: BYTE;
    counter    :    INT;
    
    // Beam class lines are restricted to 8 channels in the current design, since
    // there are no plans to use all 16. Channels 1-7 may be allocated to any other
    // beam classes so long as they are ordered least to greatest.
    // Channel 8 is reserved for full beam.
    {attribute 'pytmc' := 'pv: BeamClassOutputs
        io: i
        field: DESC Hardwire channel state'}
    {attribute 'TcLinkTo' := '[1] := TIIB[PMPS_Premp]^Channel 1^Output;
                              [2] := TIIB[PMPS_Premp]^Channel 2^Output;
                              [3] := TIIB[PMPS_Premp]^Channel 3^Output;
                              [4] := TIIB[PMPS_Premp]^Channel 4^Output;
                              
                              [5] := TIIB[PMPS_Premp]^Channel 5^Output;
                              [6] := TIIB[PMPS_Premp]^Channel 6^Output;
                              [7] := TIIB[PMPS_Premp]^Channel 7^Output;
                              [8] := TIIB[PMPS_Premp]^Channel 8^Output;'} // 8 - Full beam
    q_BC_ASSERTION_LINES    AT    %Q*    : ARRAY [1..MAX_BEAM_CLASS_LINES] OF    BOOL;
END_VAR
VAR CONSTANT
    MAX_BEAM_CLASS_LINES : BYTE := 8;
    BC_1HZ : BYTE := 1;
    BC_10HZ : BYTE := 2;
    BC_FULL : BYTE := 16;
END_VAR


// Determine BC
IF BP.nRate >= 1 THEN
    nBeamClass := BC_1HZ;
ELSIF BP.nRate >= 10 THEN
    nBeamClass := BC_10HZ;
ELSIF BP.nRate >= 120 THEN
    nBeamClass := BC_FULL;
END_IF


//Assert Beam Class
////////////////////////////////////
//0x0 = 0000 0000 0000 0000
//0x1 = 0000 0000 0000 0001
//0xF = 1111 1111 1111 1111

//Initialize BC lines to zero on every pass
FOR InitCounter := 1 TO MAX_BEAM_CLASS_LINES DO
    q_BC_ASSERTION_LINES[InitCounter] := FALSE;
END_FOR

//Set BC lines according to beam class
//A BC of 0x0 would pass over this loop, setting none of the lines high
// , as FOR loops check the initialized variable at the top to see if it's >
// than the "TO" variable.
FOR wBeamClass:=1 TO MIN(MAX_BEAM_CLASS_LINES-1, nBeamClass) DO
    q_BC_ASSERTION_LINES[wBeamClass] := TRUE;
END_FOR

q_BC_ASSERTION_LINES[8] := nBeamClass = 16; //Set channel 8 true if BC is 16

END_FUNCTION_BLOCK

// ---- MajorComponents/PMPS_MPS_Interface/FB_CTLS_Outputs.TcPOU
(*
Controls auxiliary beam class outputs.

1-3 are mapped to control the Cu beamline rate via the LCLS II MPS.

Maps beam rate requests to 1, 10, or full rate beam for Cu linac.

*)
FUNCTION_BLOCK FB_CTLS_Outputs
VAR_INPUT
    BP    :    ST_BeamParams;
END_VAR
VAR_OUTPUT
END_VAR
VAR
    {attribute 'pytmc' := 'pv: CTLSOutputs
        io: i
        field: DESC CTLS Rate Control hardwire channel state'}
    {attribute 'TcLinkTo' := '[1] := TIIB[PMPS_Premp]^Channel 9^Output;
                              [2] := TIIB[PMPS_Premp]^Channel 10^Output;
                              [3] := TIIB[PMPS_Premp]^Channel 11^Output;'}
    q_CLTS_ASSERTION_LINES    AT    %Q*    : ARRAY [1..3] OF    BOOL;  
END_VAR


// CLTS 1Hz
q_CLTS_ASSERTION_LINES[1] := BP.nRate >= 1;
// CLTS 10Hz
q_CLTS_ASSERTION_LINES[2] := BP.nRate >= 10;
// CLTS Full rate
q_CLTS_ASSERTION_LINES[3] := BP.nRate >= 120;

END_FUNCTION_BLOCK

// ---- MajorComponents/PMPS_MPS_Interface/FB_PhotonEnergyWatcher.TcPOU
(*
A. Wallace 2019-4-22
The photon energy watcher ensures the current and target photon energy is within
the arbirated bounds. Target in this case means, the calculated target photon energy
from the PVs that control the mechatronics of the undulators/ the electron energy.

If there are control PVs that match the monitor PVs, the control PVs are used to 
calculate a "target" photon energy. This is supposed to cover when the undulators/
electron energy is transitioning.

The abritrated bounds come from a simple AND of all the permitted ranges. See
the arbitrate action of the arbiter FB.

Note, this protection logic does not account for beam-off when determining fast-fault
status. If a device is requesting a limited range of eV, this request must be honored,
regardless of current beam-rate.
*)
FUNCTION_BLOCK FB_PhotonEnergyWatcher
VAR_INPUT
    i_stCurrentBeamParams    :    ST_BeamParams; //Link to global beam params
    i_stMachineTargetBeamParams    :    ST_BeamParams; //Link to global machine target beam params
    i_stRequestedBeamParams    :    ST_BeamParams; //Link to arbiter output or beam param. requestor
    // Reset fault
    i_xReset: BOOL;
END_VAR
VAR_OUTPUT
END_VAR
VAR_IN_OUT
    io_fbFFHWO    :    FB_HardwareFFOutput;
END_VAR
VAR
    xPhotonEnergyWithinBounds    :    BOOL;
    fbFF    :    FB_FastFault :=(
        i_DevName := 'ARBITER:K:PhotonEnergyWatcher',
        i_Desc := 'Fault occurs when the calculated machine photon energy (K value calculated by undulator
                    gap, and electron energy) falls outside the permitted range.',
        i_TypeCode := 16#9010);
END_VAR

xPhotonEnergyWithinBounds := (i_stCurrentBeamParams.neVRange AND i_stRequestedBeamParams.neVRange) = i_stCurrentBeamParams.neVRange;

fbFF(i_xOK := xPhotonEnergyWithinBounds,
    i_xReset := i_xReset,
    io_fbFFHWO := io_fbFFHWO);

END_FUNCTION_BLOCK

// ---- TestComponents/FB_evRangeCalculator_Test.TcPOU
{attribute 'call_after_init'}
FUNCTION_BLOCK FB_evRangeCalculator_Test EXTENDS FB_TestSuite
VAR_INPUT
END_VAR
VAR_OUTPUT
END_VAR
VAR
END_VAR

BasicFunction();

METHOD BasicFunction
VAR_INPUT
END_VAR
VAR
    LastWord : WORD := 2#0000_0000_0000_0010;
END_VAR
TEST('CheckRanges');
//Lower limit equal
AssertTrue(
    F_eVRangeCalculator(300, 0) = 2#0000_0000_0000_0100,
    'Lower limit not inclusive');
//Mid range
AssertTrue(
    F_eVRangeCalculator(251, 0) = 2#0000_0000_0000_0010,
    'In range failed, whatever you did, it broke this really bad.');
//Out of range
AssertFalse(
    F_eVRangeCalculator(300.1, 0) = 2#0000_0000_0000_0010,
    'Out of range failed, whatever you did, it broke this really bad.');

TEST_FINISHED();

TEST('Negative eV failsafes');
//Negative eV
AssertTrue(
    F_eVRangeCalculator(-300, 0) = 16#FFFF,
    'Working with antimatter? Negative eV should failsafe to FFFF.');    

TEST_FINISHED();

TEST('Check hyst keeps');

AssertTrue(
    F_eVRangeCalculator(350, 2#0000_0000_0000_0010) = 2#0000_0000_0000_0110,
    'Moving up does not stick.');
    
AssertTrue(
    F_eVRangeCalculator(150, 2#0000_0000_0000_0010) = 2#0000_0000_0000_0011,
    'Moving down does not stick.');

TEST_FINISHED();

TEST('Check hyst drops');

AssertTrue(
    F_eVRangeCalculator(351, 2#0000_0000_0000_0010) = 2#0000_0000_0000_0100,
    'Moving up does not drop.');
    
AssertTrue(
    F_eVRangeCalculator(149, 2#0000_0000_0000_0010) = 2#0000_0000_0000_0001,
    'Moving down does not drop.');

TEST_FINISHED();
END_METHOD

END_FUNCTION_BLOCK

// ---- TestComponents/FB_PhotonEnergyWatcher_Test.TcPOU
{attribute 'call_after_init'}
FUNCTION_BLOCK FB_PhotonEnergyWatcher_Test EXTENDS TcUnit.FB_TestSuite
VAR_INPUT
END_VAR
VAR_OUTPUT
END_VAR
VAR

END_VAR

PEWatcherBasicFunction();

METHOD PEWatcherBasicFunction
VAR_INPUT
END_VAR
VAR_INST
    fbPEW    :    FB_PhotonEnergyWatcher;
    fbFFO    :    FB_HardwareFFOutput;
    q_Output    :    BOOL;
    
    stCurBeamParams    :    ST_BeamParams;
    stMachineTargetBeamParams    :    ST_BeamParams;
    stReqBeamParams    :    ST_BeamParams;
END_VAR
TEST('PEWatcherBasicFunction');

//Clear FFO fault to start
fbFFO(i_xReset:=TRUE);

//All eV OK
stCurBeamParams.neVRange := F_eVRangeCalculator(800, 0);
    
stMachineTargetBeamParams.neVRange := 2#0000_0000_1000_0000;

stReqBeamParams.neVRange := 2#1111_1111_1111_1111;    

